C07272=1131.852,246.302,-68.893,-178.601,9.852,149.573
C07273=1131.856,246.053,-68.866,-178.602,9.850,149.573
C07274=1131.860,245.805,-68.838,-178.604,9.848,149.573
C07275=1131.865,245.556,-68.810,-178.605,9.846,149.572
C07276=1131.870,245.308,-68.783,-178.606,9.844,149.572
C07277=1131.874,245.060,-68.754,-178.607,9.842,149.572
C07278=1131.878,244.811,-68.727,-178.609,9.840,149.572
C07279=1131.882,244.563,-68.699,-178.610,9.837,149.572
C07280=1131.887,244.314,-68.672,-178.612,9.835,149.572
C07281=1131.891,244.066,-68.644,-178.613,9.834,149.572
C07282=1131.895,243.818,-68.616,-178.615,9.831,149.572
C07283=1131.900,243.569,-68.589,-178.617,9.829,149.571
C07284=1131.904,243.321,-68.561,-178.618,9.827,149.571
C07285=1131.909,243.072,-68.533,-178.620,9.825,149.571
C07286=1131.913,242.824,-68.506,-178.622,9.822,149.571
C07287=1131.918,242.575,-68.479,-178.623,9.820,149.571
C07288=1131.921,242.327,-68.450,-178.625,9.819,149.571
C07289=1131.926,242.078,-68.423,-178.627,9.816,149.571
C07290=1131.930,241.830,-68.396,-178.629,9.814,149.571
C07291=1131.934,241.581,-68.368,-178.631,9.812,149.571
C07292=1131.939,241.333,-68.340,-178.633,9.809,149.571
C07293=1131.943,241.085,-68.313,-178.635,9.807,149.571
C07294=1131.947,240.836,-68.285,-178.638,9.804,149.571
C07295=1131.952,240.588,-68.258,-178.639,9.802,149.571
C07296=1131.956,240.374,-68.234,-178.641,9.801,149.571
C07297=1131.959,240.159,-68.210,-178.643,9.799,149.571
C07298=1131.964,239.946,-68.186,-178.645,9.796,149.571
C07299=1131.967,239.732,-68.163,-178.647,9.794,149.571
C07300=1131.970,239.517,-68.140,-178.649,9.792,149.571
C07301=1131.974,239.303,-68.116,-178.651,9.790,149.571
C07302=1131.978,239.090,-68.093,-178.653,9.788,149.571
C07303=1131.982,238.876,-68.068,-178.656,9.786,149.571
C07304=1131.986,238.626,-68.041,-178.658,9.783,149.571
C07305=1131.991,238.378,-68.014,-178.661,9.781,149.571
C07306=1131.995,238.130,-67.986,-178.663,9.779,149.572
C07307=1132.000,237.881,-67.959,-178.665,9.775,149.572
C07308=1132.003,237.633,-67.932,-178.668,9.773,149.572
C07309=1132.008,237.385,-67.904,-178.671,9.771,149.572
C07310=1132.012,237.136,-67.877,-178.674,9.768,149.572
C07311=1132.017,236.888,-67.850,-178.677,9.765,149.572
C07312=1132.022,236.639,-67.823,-178.679,9.763,149.572
C07313=1132.025,236.391,-67.795,-178.681,9.760,149.572
C07314=1132.030,236.142,-67.768,-178.684,9.757,149.572
C07315=1132.035,235.894,-67.741,-178.687,9.755,149.572
C07316=1132.039,235.645,-67.714,-178.690,9.752,149.572
C07317=1132.043,235.397,-67.686,-178.693,9.749,149.573
C07318=1132.047,235.148,-67.659,-178.696,9.746,149.573
C07319=1132.052,234.900,-67.632,-178.700,9.743,149.573
C07320=1132.056,234.651,-67.605,-178.703,9.740,149.573
C07321=1132.061,234.403,-67.578,-178.706,9.737,149.573
C07322=1132.065,234.154,-67.551,-178.709,9.735,149.573
C07323=1132.069,233.906,-67.524,-178.713,9.732,149.574
C07324=1132.074,233.657,-67.497,-178.715,9.729,149.574
C07325=1132.078,233.409,-67.470,-178.719,9.725,149.574
C07326=1132.083,233.161,-67.442,-178.722,9.722,149.574
C07327=1132.087,232.912,-67.415,-178.726,9.719,149.574
C07328=1132.091,232.664,-67.389,-178.729,9.717,149.574
C07329=1132.095,232.415,-67.361,-178.733,9.713,149.574
C07330=1132.100,232.166,-67.334,-178.735,9.710,149.575
C07331=1132.104,231.918,-67.308,-178.739,9.707,149.575
C07332=1132.108,231.670,-67.281,-178.743,9.704,149.575
C07333=1132.113,231.421,-67.254,-178.747,9.700,149.575
C07334=1132.118,231.172,-67.227,-178.750,9.697,149.575
C07335=1132.122,230.924,-67.201,-178.753,9.694,149.575
C07336=1132.127,230.675,-67.174,-178.757,9.691,149.576
C07337=1132.131,230.427,-67.147,-178.761,9.687,149.576
C07338=1132.135,230.179,-67.120,-178.765,9.683,149.576
C07339=1132.139,229.929,-67.093,-178.769,9.680,149.576
C07340=1132.143,229.681,-67.066,-178.773,9.676,149.576
C07341=1132.148,229.432,-67.040,-178.777,9.673,149.577
C07342=1132.153,229.184,-67.013,-178.781,9.669,149.577
C07343=1132.157,228.935,-66.987,-178.784,9.665,149.577
C07344=1132.161,228.687,-66.959,-178.788,9.662,149.577
C07345=1132.166,228.438,-66.934,-178.792,9.659,149.577
C07346=1132.170,228.190,-66.907,-178.796,9.655,149.577
C07347=1132.174,227.941,-66.880,-178.799,9.652,149.578
C07348=1132.179,227.692,-66.854,-178.803,9.648,149.578
C07349=1132.184,227.444,-66.827,-178.806,9.644,149.578
C07350=1132.188,227.196,-66.800,-178.810,9.641,149.578
C07351=1132.193,226.947,-66.774,-178.813,9.637,149.578
C07352=1132.197,226.733,-66.751,-178.816,9.634,149.578
C07353=1132.200,226.519,-66.728,-178.820,9.631,149.578
C07354=1132.204,226.305,-66.705,-178.822,9.628,149.578
C07355=1132.207,226.090,-66.683,-178.825,9.625,149.578
C07356=1132.211,225.877,-66.661,-178.828,9.622,149.578
C07357=1132.215,225.662,-66.637,-178.831,9.619,149.578
C07358=1132.219,225.448,-66.615,-178.833,9.616,149.578
C07359=1132.222,225.234,-66.592,-178.836,9.614,149.578
C07360=1132.227,224.985,-66.565,-178.840,9.610,149.578
C07361=1132.231,224.736,-66.539,-178.843,9.606,149.579
C07362=1132.236,224.487,-66.513,-178.846,9.603,149.578
C07363=1132.241,224.240,-66.487,-178.849,9.600,149.579
C07364=1132.245,223.991,-66.461,-178.852,9.596,149.579
C07365=1132.250,223.742,-66.434,-178.855,9.593,149.579
C07366=1132.254,223.494,-66.408,-178.858,9.590,149.579
C07367=1132.258,223.245,-66.382,-178.861,9.586,149.578
C07368=1132.263,222.996,-66.356,-178.864,9.583,149.579
C07369=1132.267,222.747,-66.330,-178.867,9.579,149.579
C07370=1132.271,222.499,-66.303,-178.870,9.576,149.578
C07371=1132.277,222.251,-66.277,-178.873,9.572,149.578
C07372=1132.281,222.002,-66.252,-178.875,9.569,149.578
C07373=1132.285,221.754,-66.225,-178.878,9.566,149.578
C07374=1132.290,221.505,-66.199,-178.881,9.563,149.578
C07375=1132.294,221.256,-66.173,-178.884,9.560,149.578
C07376=1132.298,221.007,-66.147,-178.887,9.556,149.578
C07377=1132.303,220.760,-66.121,-178.889,9.553,149.578
C07378=1132.308,220.511,-66.095,-178.892,9.550,149.578
C07379=1132.312,220.262,-66.069,-178.894,9.547,149.578
C07380=1132.316,220.013,-66.043,-178.897,9.544,149.578
C07381=1132.320,219.765,-66.017,-178.899,9.541,149.578
C07382=1132.325,219.517,-65.992,-178.902,9.538,149.578
C07383=1132.330,219.268,-65.965,-178.904,9.534,149.578
C07384=1132.334,219.019,-65.939,-178.906,9.531,149.578
C07385=1132.338,218.770,-65.914,-178.909,9.528,149.578
C07386=1132.342,218.521,-65.888,-178.911,9.525,149.577
C07387=1132.347,218.273,-65.863,-178.913,9.523,149.577
C07388=1132.351,218.025,-65.836,-178.915,9.519,149.577
C07389=1132.356,217.776,-65.810,-178.918,9.516,149.577
C07390=1132.360,217.527,-65.784,-178.920,9.513,149.577
C07391=1132.365,217.279,-65.759,-178.922,9.511,149.577
C07392=1132.369,217.030,-65.733,-178.924,9.507,149.577
C07393=1132.374,216.781,-65.707,-178.926,9.505,149.577
C07394=1132.378,216.532,-65.681,-178.928,9.501,149.576
C07395=1132.383,216.284,-65.656,-178.930,9.499,149.576
C07396=1132.387,216.036,-65.630,-178.933,9.496,149.576
C07397=1132.391,215.787,-65.604,-178.934,9.493,149.576
C07398=1132.395,215.538,-65.579,-178.937,9.490,149.576
C07399=1132.401,215.289,-65.553,-178.938,9.487,149.576
C07400=1132.405,215.041,-65.527,-178.940,9.485,149.576
C07401=1132.409,214.792,-65.501,-178.942,9.482,149.575
C07402=1132.414,214.544,-65.476,-178.944,9.479,149.575
C07403=1132.418,214.295,-65.450,-178.946,9.477,149.575
C07404=1132.423,214.046,-65.424,-178.948,9.474,149.575
C07405=1132.427,213.797,-65.399,-178.949,9.472,149.575
C07406=1132.432,213.549,-65.373,-178.952,9.468,149.575
C07407=1132.436,213.300,-65.348,-178.953,9.466,149.575
C07408=1132.440,213.087,-65.326,-178.954,9.464,149.574
C07409=1132.443,212.872,-65.304,-178.955,9.462,149.574
C07410=1132.448,212.657,-65.281,-178.957,9.460,149.574
C07411=1132.451,212.443,-65.260,-178.958,9.458,149.574
C07412=1132.456,212.229,-65.238,-178.959,9.456,149.574
C07413=1132.459,212.014,-65.216,-178.960,9.453,149.574
C07414=1132.463,211.800,-65.194,-178.962,9.452,149.574
C07415=1132.467,211.586,-65.172,-178.963,9.449,149.574
C07416=1132.471,211.337,-65.146,-178.965,9.447,149.573
C07417=1132.476,211.088,-65.120,-178.967,9.444,149.573
C07418=1132.481,210.840,-65.095,-178.969,9.442,149.573
C07419=1132.485,210.591,-65.070,-178.970,9.439,149.573
C07420=1132.489,210.343,-65.045,-178.972,9.437,149.573
C07421=1132.493,210.094,-65.019,-178.974,9.435,149.573
C07422=1132.498,209.845,-64.994,-178.976,9.432,149.573
C07423=1132.502,209.597,-64.968,-178.978,9.430,149.573
C07424=1132.507,209.348,-64.943,-178.980,9.427,149.573
C07425=1132.511,209.099,-64.917,-178.982,9.425,149.573
C07426=1132.516,208.851,-64.892,-178.984,9.422,149.573
C07427=1132.521,208.601,-64.867,-178.987,9.419,149.573
C07428=1132.525,208.353,-64.842,-178.988,9.417,149.573
C07429=1132.530,208.104,-64.816,-178.991,9.415,149.573
C07430=1132.534,207.856,-64.790,-178.993,9.412,149.573
C07431=1132.539,207.607,-64.766,-178.995,9.410,149.573
C07432=1132.542,207.358,-64.740,-178.998,9.407,149.573
C07433=1132.547,207.110,-64.715,-179.001,9.404,149.573
C07434=1132.552,206.861,-64.690,-179.003,9.402,149.573
C07435=1132.557,206.613,-64.665,-179.006,9.399,149.573
C07436=1132.561,206.363,-64.640,-179.008,9.396,149.573
C07437=1132.565,206.115,-64.614,-179.011,9.393,149.573
C07438=1132.569,205.867,-64.589,-179.014,9.390,149.573
C07439=1132.574,205.617,-64.564,-179.016,9.387,149.573
C07440=1132.579,205.369,-64.539,-179.019,9.385,149.573
C07441=1132.583,205.120,-64.514,-179.022,9.382,149.573
C07442=1132.588,204.872,-64.488,-179.025,9.379,149.573
C07443=1132.592,204.623,-64.464,-179.028,9.376,149.573
C07444=1132.597,204.375,-64.438,-179.031,9.373,149.574
C07445=1132.601,204.125,-64.413,-179.034,9.370,149.574
C07446=1132.606,203.877,-64.388,-179.037,9.367,149.574
C07447=1132.610,203.628,-64.363,-179.040,9.364,149.574
C07448=1132.615,203.380,-64.338,-179.043,9.361,149.574
C07449=1132.619,203.130,-64.313,-179.046,9.358,149.574
C07450=1132.624,202.882,-64.288,-179.049,9.354,149.574
C07451=1132.628,202.633,-64.263,-179.052,9.352,149.574
C07452=1132.633,202.384,-64.239,-179.056,9.348,149.574
C07453=1132.637,202.136,-64.213,-179.059,9.345,149.575
C07454=1132.642,201.887,-64.189,-179.063,9.342,149.575
C07455=1132.646,201.638,-64.164,-179.066,9.339,149.575
C07456=1132.650,201.390,-64.139,-179.069,9.336,149.575
C07457=1132.655,201.141,-64.114,-179.073,9.333,149.575
C07458=1132.660,200.892,-64.089,-179.077,9.329,149.576
C07459=1132.664,200.644,-64.064,-179.080,9.326,149.576
C07460=1132.669,200.395,-64.039,-179.084,9.322,149.576
C07461=1132.673,200.146,-64.015,-179.087,9.319,149.576
C07462=1132.678,199.897,-63.990,-179.091,9.315,149.576
C07463=1132.683,199.648,-63.966,-179.095,9.312,149.576
C07464=1132.686,199.434,-63.944,-179.099,9.308,149.577
C07465=1132.690,199.220,-63.923,-179.101,9.306,149.577
C07466=1132.694,199.006,-63.902,-179.105,9.302,149.577
C07467=1132.698,198.791,-63.881,-179.108,9.299,149.577
C07468=1132.702,198.577,-63.859,-179.112,9.296,149.577
C07469=1132.706,198.362,-63.838,-179.115,9.293,149.577
C07470=1132.710,198.148,-63.817,-179.118,9.290,149.577
C07471=1132.713,197.933,-63.796,-179.122,9.286,149.578
C07472=1132.718,197.684,-63.771,-179.125,9.283,149.578
C07473=1132.722,197.436,-63.747,-179.130,9.278,149.578
C07474=1132.728,197.187,-63.722,-179.134,9.274,149.578
C07475=1132.731,196.938,-63.698,-179.138,9.271,149.578
C07476=1132.736,196.689,-63.674,-179.142,9.267,149.578
C07477=1132.741,196.441,-63.649,-179.146,9.262,149.579
C07478=1132.745,196.192,-63.625,-179.150,9.259,149.579
C07479=1132.750,195.943,-63.600,-179.151,9.256,149.579
C07480=1132.754,195.694,-63.576,-179.153,9.253,149.578
C07481=1132.759,195.446,-63.552,-179.155,9.251,149.578
C07482=1132.763,195.197,-63.527,-179.155,9.249,149.578
C07483=1132.768,194.948,-63.503,-179.157,9.246,149.578
C07484=1132.772,194.699,-63.479,-179.158,9.244,149.578
C07485=1132.777,194.450,-63.454,-179.160,9.241,149.578
C07486=1132.781,194.201,-63.430,-179.162,9.239,149.577
C07487=1132.786,193.953,-63.406,-179.164,9.236,149.577
C07488=1132.791,193.704,-63.381,-179.165,9.234,149.577
C07489=1132.794,193.455,-63.357,-179.167,9.231,149.577
C07490=1132.799,193.207,-63.333,-179.168,9.229,149.577
C07491=1132.804,192.957,-63.309,-179.170,9.226,149.577
C07492=1132.809,192.709,-63.285,-179.172,9.224,149.576
C07493=1132.813,192.461,-63.261,-179.174,9.221,149.576
C07494=1132.818,192.211,-63.236,-179.175,9.219,149.576
C07495=1132.822,191.963,-63.212,-179.177,9.216,149.576
C07496=1132.827,191.714,-63.188,-179.179,9.214,149.576
C07497=1132.831,191.465,-63.164,-179.180,9.211,149.576
C07498=1132.836,191.217,-63.140,-179.183,9.208,149.576
C07499=1132.840,190.967,-63.115,-179.185,9.206,149.576
C07500=1132.845,190.718,-63.092,-179.186,9.203,149.576
C07501=1132.850,190.470,-63.067,-179.188,9.201,149.576
C07502=1132.854,190.221,-63.043,-179.191,9.198,149.575
C07503=1132.859,189.972,-63.020,-179.193,9.195,149.575
C07504=1132.863,189.723,-62.995,-179.195,9.192,149.575
C07505=1132.867,189.475,-62.971,-179.197,9.190,149.575
C07506=1132.873,189.225,-62.947,-179.200,9.187,149.575
C07507=1132.877,188.977,-62.923,-179.201,9.184,149.575
C07508=1132.881,188.729,-62.899,-179.204,9.181,149.575
C07509=1132.886,188.479,-62.876,-179.205,9.179,149.575
C07510=1132.890,188.230,-62.851,-179.208,9.175,149.575
C07511=1132.895,187.982,-62.827,-179.210,9.173,149.575
C07512=1132.900,187.733,-62.803,-179.213,9.170,149.575
C07513=1132.904,187.484,-62.779,-179.215,9.167,149.575
C07514=1132.909,187.235,-62.756,-179.217,9.165,149.575
C07515=1132.913,186.987,-62.732,-179.220,9.162,149.575
C07516=1132.918,186.738,-62.708,-179.222,9.159,149.575
C07517=1132.923,186.489,-62.684,-179.225,9.156,149.575
C07518=1132.927,186.240,-62.659,-179.227,9.153,149.575
C07519=1132.931,185.991,-62.636,-179.230,9.149,149.575
C07520=1132.935,185.776,-62.615,-179.232,9.147,149.575
C07521=1132.939,185.563,-62.595,-179.234,9.145,149.575
C07522=1132.943,185.348,-62.575,-179.237,9.142,149.575
C07523=1132.947,185.133,-62.555,-179.239,9.140,149.575
C07524=1132.951,184.918,-62.534,-179.241,9.137,149.575
C07525=1132.955,184.704,-62.513,-179.243,9.135,149.575
C07526=1132.959,184.489,-62.492,-179.246,9.132,149.575
C07527=1132.962,184.275,-62.472,-179.248,9.129,149.575
C07528=1132.967,184.026,-62.449,-179.250,9.126,149.575
C07529=1132.972,183.776,-62.425,-179.254,9.123,149.575
C07530=1132.977,183.528,-62.401,-179.256,9.119,149.575
C07531=1132.981,183.279,-62.377,-179.259,9.116,149.575
C07532=1132.986,183.031,-62.353,-179.262,9.114,149.575
C07533=1132.991,182.782,-62.330,-179.265,9.110,149.575
C07534=1132.995,182.533,-62.307,-179.268,9.107,149.575
C07535=1132.999,182.284,-62.283,-179.271,9.104,149.575
C07536=1133.004,182.035,-62.260,-179.274,9.100,149.575
C07537=1133.008,181.786,-62.236,-179.276,9.097,149.575
C07538=1133.013,181.537,-62.213,-179.280,9.093,149.575
C07539=1133.017,181.289,-62.189,-179.282,9.090,149.575
C07540=1133.022,181.040,-62.166,-179.286,9.087,149.575
C07541=1133.027,180.791,-62.142,-179.289,9.083,149.575
C07542=1133.032,180.542,-62.119,-179.292,9.080,149.575
C07543=1133.036,180.293,-62.095,-179.295,9.076,149.575
C07544=1133.041,180.044,-62.071,-179.298,9.072,149.575
C07545=1133.045,179.795,-62.048,-179.301,9.070,149.576
C07546=1133.049,179.547,-62.025,-179.305,9.066,149.576
C07547=1133.054,179.298,-62.002,-179.308,9.062,149.576
C07548=1133.059,179.049,-61.979,-179.311,9.059,149.576
C07549=1133.064,178.800,-61.956,-179.313,9.056,149.575
C07550=1133.069,178.551,-61.932,-179.315,9.053,149.575
C07551=1133.073,178.303,-61.908,-179.317,9.050,149.575
C07552=1133.077,178.054,-61.885,-179.319,9.048,149.575
C07553=1133.082,177.805,-61.862,-179.321,9.044,149.575
C07554=1133.086,177.556,-61.839,-179.324,9.041,149.575
C07555=1133.091,177.307,-61.815,-179.325,9.039,149.575
C07556=1133.096,177.058,-61.792,-179.328,9.036,149.575
C07557=1133.100,176.809,-61.769,-179.330,9.032,149.575
C07558=1133.104,176.560,-61.746,-179.332,9.030,149.575
C07559=1133.109,176.311,-61.722,-179.334,9.027,149.574
C07560=1133.114,176.063,-61.700,-179.337,9.024,149.574
C07561=1133.118,175.814,-61.677,-179.338,9.021,149.574
C07562=1133.123,175.565,-61.653,-179.341,9.018,149.574
C07563=1133.128,175.316,-61.630,-179.343,9.015,149.574
C07564=1133.132,175.067,-61.608,-179.345,9.012,149.574
C07565=1133.137,174.818,-61.585,-179.347,9.009,149.574
C07566=1133.142,174.569,-61.561,-179.350,9.006,149.574
C07567=1133.147,174.320,-61.538,-179.351,9.003,149.574
C07568=1133.151,174.072,-61.515,-179.354,9.000,149.574
C07569=1133.155,173.823,-61.492,-179.356,8.997,149.574
C07570=1133.160,173.574,-61.469,-179.359,8.994,149.573
C07571=1133.164,173.325,-61.446,-179.360,8.991,149.573
C07572=1133.169,173.075,-61.423,-179.363,8.988,149.573
C07573=1133.174,172.827,-61.400,-179.365,8.985,149.573
C07574=1133.178,172.578,-61.378,-179.368,8.982,149.573
C07575=1133.183,172.329,-61.354,-179.369,8.979,149.573
C07576=1133.188,172.089,-61.332,-179.372,8.976,149.573
C07577=1133.192,171.850,-61.310,-179.374,8.973,149.573
C07578=1133.196,171.610,-61.288,-179.376,8.970,149.573
C07579=1133.201,171.370,-61.266,-179.378,8.967,149.573
C07580=1133.206,171.132,-61.245,-179.381,8.964,149.573
C07581=1133.210,170.892,-61.223,-179.383,8.961,149.573
C07582=1133.214,170.652,-61.201,-179.385,8.958,149.572
C07583=1133.219,170.413,-61.179,-179.387,8.955,149.572
C07584=1133.241,169.216,-61.071,-178.557,7.312,148.954
C07585=1133.249,168.816,-61.036,-178.561,7.308,148.954
C07586=1133.253,168.568,-61.014,-178.565,7.306,148.955
C07587=1133.257,168.318,-60.992,-178.567,7.304,148.955
C07588=1133.263,168.070,-60.969,-178.570,7.301,148.955
C07589=1133.267,167.821,-60.947,-178.573,7.300,148.956
C07590=1133.271,167.571,-60.924,-178.576,7.297,148.956
C07591=1133.277,167.323,-60.902,-178.578,7.295,148.956
C07592=1133.281,167.073,-60.880,-178.582,7.292,148.957
C07593=1133.286,166.825,-60.858,-178.584,7.291,148.957
C07594=1133.290,166.576,-60.836,-178.587,7.288,148.957
C07595=1133.296,166.327,-60.813,-178.590,7.286,148.957
C07596=1133.300,166.078,-60.791,-178.593,7.283,148.958
C07597=1133.305,165.829,-60.770,-178.596,7.282,148.958
C07598=1133.309,165.580,-60.748,-178.599,7.279,148.958
C07599=1133.314,165.332,-60.725,-178.602,7.277,148.959
C07600=1133.319,165.082,-60.703,-178.604,7.274,148.959
C07601=1133.323,164.833,-60.681,-178.607,7.273,148.959
C07602=1133.328,164.584,-60.659,-178.610,7.270,148.960
C07603=1133.333,164.335,-60.637,-178.613,7.268,148.960
C07604=1133.337,164.086,-60.615,-178.616,7.266,148.960
C07605=1133.342,163.837,-60.593,-178.619,7.264,148.960
C07606=1133.347,163.588,-60.571,-178.621,7.262,148.961
C07607=1133.352,163.339,-60.549,-178.624,7.259,148.961
C07608=1133.356,163.090,-60.527,-178.627,7.258,148.961
C07609=1133.361,162.841,-60.505,-178.630,7.255,148.961
C07610=1133.365,162.592,-60.483,-178.632,7.253,148.962
C07611=1133.370,162.343,-60.462,-178.636,7.251,148.962
C07612=1133.374,162.094,-60.440,-178.638,7.249,148.962
C07613=1133.379,161.845,-60.418,-178.641,7.246,148.963
C07614=1133.384,161.595,-60.395,-178.644,7.244,148.963
C07615=1133.389,161.347,-60.374,-178.647,7.242,148.963
C07616=1133.393,161.097,-60.352,-178.650,7.240,148.964
C07617=1133.398,160.849,-60.330,-178.652,7.238,148.964
C07618=1133.403,160.600,-60.308,-178.656,7.235,148.964
C07619=1133.407,160.351,-60.286,-178.658,7.233,148.964
C07620=1133.412,160.102,-60.264,-178.661,7.231,148.965
C07621=1133.416,159.853,-60.242,-178.664,7.229,148.965
C07622=1133.421,159.604,-60.221,-178.667,7.227,148.966
C07623=1133.426,159.356,-60.199,-178.669,7.225,148.966
C07624=1133.431,159.106,-60.178,-178.672,7.223,148.966
C07625=1133.435,158.857,-60.156,-178.675,7.220,148.966
C07626=1133.440,158.608,-60.134,-178.678,7.218,148.967
C07627=1133.445,158.359,-60.112,-178.681,7.216,148.967
C07628=1133.449,158.110,-60.091,-178.684,7.214,148.967
C07629=1133.454,157.860,-60.069,-178.687,7.212,148.968
C07630=1133.458,157.592,-60.046,-178.690,7.210,148.968
C07631=1133.464,157.323,-60.022,-178.692,7.207,148.968
C07632=1133.469,157.053,-60.000,-178.696,7.205,148.969
C07633=1133.474,156.785,-59.976,-178.698,7.203,148.969
C07634=1133.479,156.536,-59.954,-178.702,7.200,148.969
C07635=1133.484,156.287,-59.933,-178.704,7.199,148.970
C07636=1133.488,156.038,-59.911,-178.707,7.197,148.970
C07637=1133.493,155.789,-59.889,-178.710,7.194,148.970
C07638=1133.498,155.540,-59.869,-178.713,7.192,148.971
C07639=1133.502,155.291,-59.847,-178.716,7.190,148.971
C07640=1133.507,155.042,-59.825,-178.718,7.188,148.971
C07641=1133.512,154.793,-59.804,-178.721,7.186,148.972
C07642=1133.517,154.544,-59.783,-178.724,7.184,148.972
C07643=1133.521,154.294,-59.761,-178.727,7.182,148.972
C07644=1133.526,154.045,-59.740,-178.730,7.179,148.972
C07645=1133.530,153.797,-59.718,-178.733,7.177,148.973
C07646=1133.535,153.547,-59.697,-178.735,7.176,148.973
C07647=1133.540,153.299,-59.675,-178.739,7.173,148.974
C07648=1133.545,153.049,-59.654,-178.741,7.171,148.974
C07649=1133.550,152.801,-59.633,-178.744,7.169,148.974
C07650=1133.554,152.551,-59.612,-178.747,7.167,148.975
C07651=1133.558,152.302,-59.590,-178.750,7.165,148.975
C07652=1133.564,152.053,-59.569,-178.753,7.163,148.975
C07653=1133.569,151.804,-59.548,-178.755,7.160,148.975
C07654=1133.573,151.554,-59.526,-178.758,7.159,148.976
C07655=1133.577,151.306,-59.505,-178.761,7.156,148.976
C07656=1133.582,151.057,-59.484,-178.764,7.155,148.977
C07657=1133.587,150.808,-59.463,-178.767,7.153,148.977
C07658=1133.592,150.559,-59.442,-178.769,7.150,148.977
C07659=1133.596,150.309,-59.421,-178.772,7.148,148.977
C07660=1133.601,150.061,-59.399,-178.775,7.147,148.978
C07661=1133.606,149.811,-59.378,-178.778,7.144,148.978
C07662=1133.610,149.563,-59.357,-178.781,7.142,148.979
C07663=1133.616,149.314,-59.336,-178.784,7.140,148.979
C07664=1133.621,149.065,-59.315,-178.786,7.138,148.979
C07665=1133.624,148.816,-59.294,-178.789,7.136,148.980
C07666=1133.629,148.566,-59.273,-178.792,7.134,148.980
C07667=1133.635,148.317,-59.252,-178.795,7.132,148.980
C07668=1133.639,148.069,-59.231,-178.797,7.130,148.980
C07669=1133.644,147.819,-59.210,-178.801,7.127,148.981
C07670=1133.649,147.570,-59.189,-178.803,7.126,148.981
C07671=1133.653,147.321,-59.167,-178.806,7.124,148.982
C07672=1133.658,147.072,-59.146,-178.809,7.121,148.982
C07673=1133.662,146.823,-59.126,-178.812,7.119,148.982
C07674=1133.667,146.574,-59.105,-178.814,7.118,148.983
C07675=1133.673,146.324,-59.084,-178.817,7.116,148.983
C07676=1133.677,146.076,-59.063,-178.820,7.113,148.983
C07677=1133.682,145.827,-59.042,-178.823,7.112,148.984
C07678=1133.686,145.578,-59.022,-178.826,7.110,148.984
C07679=1133.691,145.328,-59.000,-178.829,7.107,148.984
C07680=1133.695,145.079,-58.980,-178.831,7.106,148.985
C07681=1133.700,144.830,-58.958,-178.834,7.104,148.985
C07682=1133.705,144.581,-58.937,-178.838,7.101,148.985
C07683=1133.710,144.332,-58.917,-178.840,7.100,148.986
C07684=1133.715,144.083,-58.896,-178.843,7.098,148.986
C07685=1133.719,143.834,-58.876,-178.846,7.095,148.986
C07686=1133.725,143.585,-58.855,-178.849,7.093,148.987
C07687=1133.729,143.336,-58.834,-178.851,7.092,148.987
C07688=1133.734,143.087,-58.814,-178.854,7.090,148.987
C07689=1133.739,142.837,-58.793,-178.857,7.087,148.988
C07690=1133.743,142.589,-58.773,-178.860,7.086,148.988
C07691=1133.748,142.339,-58.752,-178.863,7.084,148.989
C07692=1133.753,142.090,-58.731,-178.866,7.081,148.989
C07693=1133.757,141.841,-58.709,-178.868,7.079,148.989
C07694=1133.761,141.592,-58.689,-178.871,7.078,148.990
C07695=1133.767,141.342,-58.669,-178.874,7.076,148.990
C07696=1133.771,141.093,-58.648,-178.877,7.074,148.990
C07697=1133.776,140.844,-58.628,-178.880,7.072,148.991
C07698=1133.781,140.595,-58.607,-178.882,7.070,148.991
C07699=1133.785,140.346,-58.586,-178.885,7.067,148.991
C07700=1133.791,140.097,-58.566,-178.888,7.066,148.992
C07701=1133.795,139.848,-58.545,-178.891,7.064,148.992
C07702=1133.799,139.599,-58.525,-178.893,7.062,148.992
C07703=1133.805,139.350,-58.504,-178.897,7.060,148.993
C07704=1133.809,139.101,-58.483,-178.899,7.058,148.993
C07705=1133.814,138.852,-58.463,-178.902,7.056,148.994
C07706=1133.819,138.603,-58.442,-178.905,7.055,148.994
C07707=1133.824,138.354,-58.423,-178.908,7.052,148.994
C07708=1133.828,138.105,-58.402,-178.910,7.050,148.995
C07709=1133.834,137.855,-58.381,-178.913,7.048,148.995
C07710=1133.838,137.606,-58.361,-178.916,7.047,148.995
C07711=1133.843,137.358,-58.341,-178.919,7.044,148.996
C07712=1133.848,137.108,-58.320,-178.922,7.043,148.996
C07713=1133.852,136.859,-58.300,-178.925,7.041,148.996
C07714=1133.857,136.610,-58.280,-178.927,7.039,148.997
C07715=1133.861,136.361,-58.259,-178.931,7.037,148.997
C07716=1133.867,136.112,-58.238,-178.933,7.035,148.997
C07717=1133.871,135.862,-58.219,-178.936,7.033,148.998
C07718=1133.876,135.613,-58.198,-178.938,7.031,148.998
C07719=1133.880,135.364,-58.178,-178.942,7.029,148.999
C07720=1133.886,135.115,-58.158,-178.944,7.027,148.999
C07721=1133.891,134.866,-58.138,-178.947,7.025,148.999
C07722=1133.895,134.617,-58.117,-178.950,7.024,149.000
C07723=1133.900,134.367,-58.098,-178.953,7.021,149.000
C07724=1133.904,134.118,-58.077,-178.956,7.019,149.001
C07725=1133.909,133.869,-58.056,-178.959,7.018,149.001
C07726=1133.914,133.620,-58.037,-178.961,7.016,149.001
C07727=1133.919,133.371,-58.016,-178.964,7.014,149.002
C07728=1133.924,133.122,-57.997,-178.967,7.012,149.002
C07729=1133.928,132.873,-57.977,-178.970,7.010,149.002
C07730=1133.933,132.624,-57.956,-178.972,7.008,149.003
C07731=1133.938,132.374,-57.936,-178.975,7.006,149.003
C07732=1133.943,132.125,-57.916,-178.978,7.005,149.004
C07733=1133.947,131.876,-57.896,-178.981,7.002,149.004
C07734=1133.952,131.608,-57.874,-178.984,7.001,149.004
C07735=1133.958,131.339,-57.853,-178.987,6.998,149.005
C07736=1133.963,131.071,-57.832,-178.990,6.996,149.005
C07737=1133.969,130.802,-57.809,-178.993,6.995,149.005
C07738=1133.973,130.553,-57.790,-178.996,6.992,149.006
C07739=1133.978,130.304,-57.769,-178.999,6.991,149.006
C07740=1133.983,130.054,-57.750,-179.001,6.989,149.007
C07741=1133.987,129.805,-57.730,-179.004,6.987,149.007
C07742=1133.992,129.556,-57.710,-179.007,6.985,149.007
C07743=1133.997,129.307,-57.690,-179.010,6.983,149.008
C07744=1134.002,129.058,-57.670,-179.013,6.981,149.008
C07745=1134.006,128.808,-57.650,-179.016,6.980,149.009
C07746=1134.012,128.559,-57.631,-179.018,6.978,149.009
C07747=1134.016,128.310,-57.611,-179.021,6.976,149.009
C07748=1134.021,128.061,-57.591,-179.024,6.975,149.010
C07749=1134.025,127.812,-57.571,-179.027,6.972,149.010
C07750=1134.031,127.563,-57.551,-179.030,6.970,149.011
C07751=1134.035,127.314,-57.532,-179.033,6.969,149.011
C07752=1134.040,127.065,-57.511,-179.035,6.967,149.011
C07753=1134.044,126.815,-57.492,-179.038,6.965,149.012
C07754=1134.050,126.566,-57.472,-179.040,6.963,149.012
C07755=1134.055,126.317,-57.453,-179.044,6.961,149.012
C07756=1134.059,126.068,-57.432,-179.046,6.959,149.013
C07757=1134.064,125.819,-57.413,-179.049,6.957,149.013
C07758=1134.069,125.569,-57.393,-179.052,6.956,149.014
C07759=1134.074,125.320,-57.374,-179.055,6.954,149.014
C07760=1134.078,125.072,-57.354,-179.057,6.952,149.014
C07761=1134.083,124.822,-57.335,-179.060,6.951,149.015
C07762=1134.088,124.573,-57.315,-179.063,6.948,149.015
C07763=1134.092,124.323,-57.295,-179.066,6.946,149.016
C07764=1134.097,124.075,-57.275,-179.069,6.945,149.016
C07765=1134.102,123.825,-57.256,-179.072,6.943,149.016
C07766=1134.107,123.576,-57.236,-179.074,6.941,149.017
C07767=1134.112,123.327,-57.217,-179.077,6.940,149.017
C07768=1134.116,123.077,-57.198,-179.080,6.938,149.018
C07769=1134.122,122.829,-57.178,-179.083,6.936,149.018
C07770=1134.126,122.579,-57.159,-179.086,6.934,149.018
C07771=1134.131,122.329,-57.139,-179.088,6.932,149.019
C07772=1134.136,122.081,-57.119,-179.091,6.930,149.019
C07773=1134.141,121.832,-57.099,-179.094,6.929,149.020
C07774=1134.145,121.582,-57.080,-179.097,6.927,149.020
C07775=1134.150,121.334,-57.061,-179.099,6.925,149.020
C07776=1134.155,121.084,-57.041,-179.102,6.924,149.021
C07777=1134.160,120.835,-57.022,-179.105,6.921,149.021
C07778=1134.164,120.586,-57.003,-179.108,6.920,149.022
C07779=1134.169,120.336,-56.983,-179.111,6.918,149.022
C07780=1134.174,120.087,-56.964,-179.114,6.916,149.022
C07781=1134.179,119.838,-56.945,-179.116,6.915,149.023
C07782=1134.184,119.589,-56.926,-179.119,6.913,149.023
C07783=1134.188,119.340,-56.906,-179.122,6.911,149.024
C07784=1134.193,119.090,-56.887,-179.125,6.909,149.024
C07785=1134.199,118.841,-56.867,-179.127,6.908,149.024
C07786=1134.203,118.592,-56.848,-179.131,6.905,149.025
C07787=1134.208,118.343,-56.829,-179.133,6.904,149.025
C07788=1134.213,118.093,-56.810,-179.136,6.902,149.026
C07789=1134.218,117.844,-56.791,-179.139,6.900,149.026
C07790=1134.222,117.595,-56.772,-179.142,6.899,149.026
C07791=1134.228,117.346,-56.752,-179.144,6.897,149.027
C07792=1134.232,117.097,-56.733,-179.147,6.895,149.027
C07793=1134.237,116.848,-56.714,-179.150,6.894,149.028
C07794=1134.242,116.598,-56.694,-179.152,6.892,149.028
C07795=1134.247,116.349,-56.676,-179.155,6.890,149.028
C07796=1134.251,116.100,-56.657,-179.158,6.889,149.029
C07797=1134.257,115.851,-56.637,-179.161,6.887,149.029
C07798=1134.261,115.601,-56.618,-179.164,6.884,149.030
C07799=1134.266,115.353,-56.599,-179.167,6.883,149.030
C07800=1134.271,115.102,-56.580,-179.169,6.881,149.030
C07801=1134.276,114.854,-56.561,-179.172,6.879,149.031
C07802=1134.280,114.604,-56.542,-179.175,6.878,149.031
C07803=1134.285,114.356,-56.523,-179.178,6.876,149.032
C07804=1134.290,114.105,-56.504,-179.180,6.874,149.032
C07805=1134.295,113.857,-56.485,-179.183,6.873,149.032
C07806=1134.299,113.607,-56.466,-179.186,6.871,149.033
C07807=1134.305,113.358,-56.446,-179.189,6.870,149.034
C07808=1134.309,113.109,-56.428,-179.192,6.868,149.034
C07809=1134.314,112.860,-56.409,-179.194,6.866,149.034
C07810=1134.319,112.611,-56.390,-179.197,6.865,149.035
C07811=1134.324,112.361,-56.371,-179.200,6.863,149.035
C07812=1134.329,112.112,-56.352,-179.203,6.861,149.036
C07813=1134.334,111.862,-56.334,-179.205,6.860,149.036
C07814=1134.338,111.614,-56.315,-179.208,6.858,149.036
C07815=1134.344,111.365,-56.296,-179.211,6.856,149.037
C07816=1134.348,111.115,-56.277,-179.214,6.854,149.037
C07817=1134.353,110.866,-56.258,-179.217,6.852,149.038
C07818=1134.358,110.616,-56.240,-179.220,6.850,149.038
C07819=1134.363,110.367,-56.220,-179.222,6.849,149.038
C07820=1134.368,110.119,-56.202,-179.225,6.847,149.039
C07821=1134.373,109.869,-56.183,-179.228,6.845,149.039
C07822=1134.377,109.620,-56.164,-179.231,6.844,149.040
C07823=1134.382,109.370,-56.146,-179.233,6.842,149.040
C07824=1134.387,109.121,-56.126,-179.236,6.840,149.040
C07825=1134.392,108.872,-56.108,-179.239,6.839,149.041
C07826=1134.397,108.623,-56.089,-179.242,6.837,149.042
C07827=1134.402,108.373,-56.071,-179.245,6.836,149.042
C07828=1134.406,108.125,-56.052,-179.247,6.834,149.042
C07829=1134.411,107.875,-56.033,-179.250,6.832,149.043
C07830=1134.416,107.625,-56.015,-179.253,6.831,149.043
C07831=1134.421,107.377,-55.996,-179.256,6.829,149.044
C07832=1134.426,107.127,-55.977,-179.258,6.827,149.044
C07833=1134.430,106.878,-55.959,-179.261,6.826,149.044
C07834=1134.436,106.629,-55.940,-179.264,6.824,149.045
C07835=1134.440,106.379,-55.922,-179.267,6.822,149.045
C07836=1134.445,106.130,-55.903,-179.269,6.821,149.046
C07837=1134.451,105.881,-55.885,-179.272,6.819,149.046
C07838=1134.455,105.612,-55.865,-179.275,6.818,149.047
C07839=1134.460,105.344,-55.845,-179.278,6.816,149.047
C07840=1134.466,105.076,-55.825,-179.281,6.813,149.047
C07841=1134.471,104.807,-55.805,-179.284,6.812,149.048
C07842=1134.476,104.558,-55.787,-179.287,6.810,149.048
C07843=1134.480,104.309,-55.768,-179.290,6.809,149.049
C07844=1134.485,104.059,-55.750,-179.293,6.807,149.049
C07845=1134.490,103.810,-55.732,-179.296,6.805,149.050
C07846=1134.496,103.561,-55.712,-179.298,6.804,149.050
C07847=1134.500,103.311,-55.694,-179.301,6.802,149.051
C07848=1134.505,103.062,-55.676,-179.304,6.800,149.051
C07849=1134.510,102.813,-55.658,-179.307,6.799,149.051
C07850=1134.515,102.564,-55.639,-179.309,6.797,149.052
C07851=1134.519,102.314,-55.620,-179.312,6.795,149.052
C07852=1134.524,102.065,-55.602,-179.314,6.795,149.053
C07853=1134.529,101.816,-55.584,-179.317,6.793,149.053
C07854=1134.534,101.567,-55.566,-179.320,6.792,149.054
C07855=1134.539,101.317,-55.548,-179.323,6.790,149.054
C07856=1134.544,101.067,-55.530,-179.326,6.788,149.055
C07857=1134.549,100.819,-55.511,-179.328,6.787,149.055
C07858=1134.554,100.570,-55.493,-179.331,6.785,149.055
C07859=1134.558,100.321,-55.475,-179.334,6.783,149.056
C07860=1134.563,100.071,-55.457,-179.336,6.782,149.056
C07861=1134.568,99.821,-55.438,-179.339,6.780,149.057
C07862=1134.573,99.572,-55.420,-179.342,6.778,149.057
C07863=1134.578,99.323,-55.402,-179.345,6.777,149.058
C07864=1134.583,99.074,-55.384,-179.348,6.775,149.058
C07865=1134.588,98.825,-55.366,-179.351,6.774,149.059
C07866=1134.592,98.575,-55.348,-179.353,6.772,149.059
C07867=1134.597,98.325,-55.330,-179.356,6.770,149.059
C07868=1134.602,98.076,-55.312,-179.359,6.769,149.060
C07869=1134.607,97.827,-55.294,-179.362,6.767,149.060
C07870=1134.612,97.578,-55.276,-179.364,6.765,149.061
C07871=1134.617,97.329,-55.258,-179.367,6.765,149.061
C07872=1134.623,97.079,-55.239,-179.370,6.763,149.062
C07873=1134.627,96.829,-55.221,-179.372,6.761,149.062
C07874=1134.632,96.580,-55.203,-179.375,6.760,149.063
C07875=1134.637,96.331,-55.185,-179.378,6.758,149.063
C07876=1134.642,96.082,-55.167,-179.381,6.756,149.063
C07877=1134.647,95.833,-55.149,-179.383,6.755,149.064
C07878=1134.651,95.584,-55.131,-179.386,6.753,149.064
C07879=1134.656,95.334,-55.113,-179.389,6.752,149.065
C07880=1134.661,95.085,-55.095,-179.392,6.750,149.065
C07881=1134.666,94.836,-55.077,-179.395,6.748,149.066
C07882=1134.671,94.587,-55.059,-179.398,6.747,149.066
C07883=1134.676,94.336,-55.041,-179.400,6.746,149.067
C07884=1134.681,94.087,-55.023,-179.402,6.744,149.067
C07885=1134.686,93.838,-55.005,-179.405,6.743,149.067
C07886=1134.690,93.589,-54.987,-179.408,6.741,149.068
C07887=1134.695,93.340,-54.970,-179.411,6.740,149.068
C07888=1134.700,93.091,-54.952,-179.414,6.738,149.069
C07889=1134.705,92.841,-54.935,-179.417,6.736,149.069
C07890=1134.710,92.592,-54.917,-179.419,6.735,149.070
C07891=1134.715,92.343,-54.899,-179.422,6.733,149.070
C07892=1134.720,92.093,-54.881,-179.425,6.731,149.071
C07893=1134.725,91.844,-54.864,-179.428,6.731,149.071
C07894=1134.730,91.594,-54.846,-179.430,6.729,149.072
C07895=1134.735,91.345,-54.828,-179.433,6.728,149.072
C07896=1134.739,91.096,-54.810,-179.436,6.726,149.072
C07897=1134.745,90.846,-54.792,-179.438,6.724,149.073
C07898=1134.749,90.597,-54.775,-179.441,6.723,149.073
C07899=1134.754,90.348,-54.757,-179.444,6.721,149.074
C07900=1134.759,90.098,-54.740,-179.447,6.720,149.074
C07901=1134.764,89.849,-54.722,-179.449,6.719,149.075
C07902=1134.769,89.600,-54.704,-179.452,6.717,149.075
C07903=1134.774,89.350,-54.687,-179.455,6.715,149.076
C07904=1134.778,89.101,-54.669,-179.458,6.714,149.076
C07905=1134.783,88.852,-54.651,-179.460,6.712,149.076
C07906=1134.788,88.603,-54.634,-179.464,6.711,149.077
C07907=1134.793,88.353,-54.616,-179.466,6.709,149.078
C07908=1134.798,88.104,-54.599,-179.469,6.707,149.078
C07909=1134.803,87.855,-54.581,-179.471,6.707,149.078
C07910=1134.808,87.605,-54.564,-179.474,6.705,149.079
C07911=1134.813,87.356,-54.546,-179.477,6.703,149.079
C07912=1134.818,87.107,-54.528,-179.480,6.702,149.080
C07913=1134.822,86.857,-54.511,-179.483,6.700,149.080
C07914=1134.827,86.608,-54.493,-179.485,6.699,149.081
C07915=1134.833,86.359,-54.477,-179.488,6.698,149.081
C07916=1134.838,86.110,-54.459,-179.490,6.696,149.082
C07917=1134.842,85.860,-54.442,-179.493,6.695,149.082
C07918=1134.847,85.611,-54.424,-179.496,6.693,149.083
C07919=1134.852,85.361,-54.407,-179.499,6.692,149.083
C07920=1134.857,85.112,-54.389,-179.502,6.690,149.083
C07921=1134.862,84.862,-54.372,-179.504,6.688,149.084
C07922=1134.867,84.613,-54.355,-179.507,6.687,149.084
C07923=1134.872,84.364,-54.337,-179.510,6.686,149.085
C07924=1134.876,84.114,-54.320,-179.513,6.684,149.085
C07925=1134.882,83.866,-54.302,-179.515,6.683,149.086
C07926=1134.887,83.616,-54.285,-179.518,6.681,149.086
C07927=1134.892,83.366,-54.269,-179.520,6.680,149.087
C07928=1134.897,83.117,-54.251,-179.523,6.679,149.087
C07929=1134.902,82.867,-54.233,-179.526,6.677,149.088
C07930=1134.906,82.618,-54.216,-179.529,6.676,149.088
C07931=1134.911,82.369,-54.199,-179.532,6.674,149.089
C07932=1134.916,82.120,-54.182,-179.534,6.672,149.089
C07933=1134.921,81.871,-54.164,-179.537,6.672,149.090
C07934=1134.926,81.621,-54.147,-179.540,6.670,149.090
C07935=1134.931,81.371,-54.130,-179.543,6.669,149.091
C07936=1134.936,81.122,-54.113,-179.545,6.667,149.091
C07937=1134.940,80.873,-54.096,-179.548,6.665,149.091
C07938=1134.946,80.624,-54.079,-179.551,6.665,149.092
C07939=1134.951,80.374,-54.062,-179.553,6.663,149.093
C07940=1134.955,80.125,-54.044,-179.556,6.661,149.093
C07941=1134.961,79.875,-54.027,-179.559,6.660,149.093
C07942=1134.966,79.607,-54.009,-179.562,6.658,149.094
C07943=1134.971,79.338,-53.991,-179.565,6.657,149.094
C07944=1134.976,79.070,-53.972,-179.568,6.655,149.095
C07945=1134.982,78.802,-53.954,-179.571,6.654,149.096
C07946=1134.987,78.552,-53.937,-179.574,6.652,149.096
C07947=1134.992,78.302,-53.920,-179.576,6.651,149.096
C07948=1134.997,78.054,-53.903,-179.578,6.650,149.097
C07949=1135.002,77.804,-53.886,-179.581,6.648,149.097
C07950=1135.007,77.555,-53.869,-179.584,6.647,149.098
C07951=1135.011,77.305,-53.852,-179.587,6.646,149.098
C07952=1135.017,77.056,-53.835,-179.589,6.644,149.099
C07953=1135.022,76.807,-53.818,-179.592,6.643,149.099
C07954=1135.026,76.557,-53.802,-179.595,6.641,149.100
C07955=1135.031,76.307,-53.784,-179.598,6.640,149.100
C07956=1135.036,76.059,-53.767,-179.600,6.639,149.101
C07957=1135.041,75.809,-53.750,-179.603,6.637,149.101
C07958=1135.046,75.560,-53.734,-179.606,6.636,149.102
C07959=1135.051,75.310,-53.716,-179.609,6.634,149.102
C07960=1135.056,75.061,-53.700,-179.611,6.633,149.103
C07961=1135.061,74.812,-53.683,-179.614,6.632,149.103
C07962=1135.066,74.562,-53.666,-179.617,6.630,149.104
C07963=1135.071,74.313,-53.650,-179.619,6.629,149.104
C07964=1135.076,74.063,-53.632,-179.622,6.628,149.105
C07965=1135.081,73.814,-53.616,-179.625,6.626,149.105
C07966=1135.086,73.565,-53.599,-179.627,6.625,149.105
C07967=1135.091,73.315,-53.582,-179.630,6.623,149.106
C07968=1135.095,73.066,-53.566,-179.633,6.623,149.107
C07969=1135.100,72.817,-53.549,-179.636,6.621,149.107
C07970=1135.106,72.567,-53.532,-179.638,6.619,149.107
C07971=1135.110,72.318,-53.515,-179.641,6.618,149.108
C07972=1135.116,72.068,-53.500,-179.644,6.617,149.109
C07973=1135.121,71.819,-53.482,-179.646,6.616,149.109
C07974=1135.125,71.569,-53.466,-179.649,6.614,149.109
C07975=1135.130,71.320,-53.450,-179.652,6.612,149.110
C07976=1135.136,71.071,-53.432,-179.654,6.611,149.110
C07977=1135.140,70.821,-53.416,-179.657,6.610,149.111
C07978=1135.145,70.572,-53.399,-179.660,6.608,149.111
C07979=1135.150,70.323,-53.382,-179.662,6.608,149.112
C07980=1135.156,70.073,-53.366,-179.665,6.606,149.112
C07981=1135.160,69.824,-53.350,-179.668,6.605,149.113
C07982=1135.165,69.574,-53.333,-179.671,6.603,149.113
C07983=1135.170,69.325,-53.316,-179.673,6.602,149.114
C07984=1135.175,69.076,-53.300,-179.676,6.601,149.114
C07985=1135.180,68.826,-53.284,-179.679,6.599,149.115
C07986=1135.185,68.577,-53.267,-179.681,6.598,149.115
C07987=1135.190,68.327,-53.250,-179.684,6.597,149.116
C07988=1135.195,68.078,-53.234,-179.687,6.595,149.116
C07989=1135.200,67.828,-53.218,-179.690,6.594,149.117
C07990=1135.205,67.579,-53.201,-179.692,6.593,149.117
C07991=1135.209,67.330,-53.185,-179.695,6.591,149.118
C07992=1135.215,67.081,-53.168,-179.698,6.590,149.118
C07993=1135.220,66.831,-53.152,-179.700,6.589,149.119
C07994=1135.225,66.581,-53.135,-179.703,6.588,149.119
C07995=1135.230,66.332,-53.119,-179.706,6.586,149.120
C07996=1135.234,66.082,-53.103,-179.708,6.585,149.120
C07997=1135.239,65.833,-53.087,-179.711,6.584,149.121
C07998=1135.244,65.584,-53.070,-179.714,6.582,149.121
C07999=1135.250,65.334,-53.054,-179.716,6.581,149.122
C08000=1135.255,65.085,-53.037,-179.719,6.580,149.122
C08001=1135.260,64.836,-53.021,-179.722,6.578,149.123
C08002=1135.264,64.586,-53.005,-179.725,6.577,149.123
C08003=1135.270,64.337,-52.989,-179.727,6.576,149.124
C08004=1135.274,64.087,-52.973,-179.730,6.574,149.124
C08005=1135.279,63.838,-52.956,-179.733,6.573,149.125
C08006=1135.284,63.589,-52.940,-179.735,6.572,149.125
C08007=1135.289,63.339,-52.924,-179.738,6.571,149.126
C08008=1135.294,63.090,-52.907,-179.741,6.569,149.126
C08009=1135.299,62.840,-52.892,-179.743,6.568,149.127
C08010=1135.304,62.591,-52.875,-179.746,6.567,149.127
C08011=1135.310,62.341,-52.859,-179.749,6.565,149.128
C08012=1135.314,62.092,-52.842,-179.751,6.564,149.128
C08013=1135.320,61.842,-52.827,-179.754,6.563,149.129
C08014=1135.324,61.593,-52.810,-179.757,6.561,149.129
C08015=1135.329,61.343,-52.794,-179.759,6.561,149.129
C08016=1135.334,61.094,-52.778,-179.762,6.559,149.130
C08017=1135.339,60.845,-52.762,-179.765,6.558,149.131
C08018=1135.344,60.596,-52.746,-179.767,6.557,149.131
C08019=1135.349,60.346,-52.730,-179.770,6.555,149.131
C08020=1135.354,60.097,-52.714,-179.773,6.555,149.132
C08021=1135.359,59.847,-52.698,-179.775,6.553,149.133
C08022=1135.364,59.597,-52.682,-179.778,6.551,149.133
C08023=1135.369,59.348,-52.665,-179.780,6.551,149.133
C08024=1135.374,59.098,-52.650,-179.784,6.549,149.134
C08025=1135.379,58.850,-52.634,-179.786,6.548,149.135
C08026=1135.384,58.600,-52.618,-179.788,6.547,149.135
C08027=1135.389,58.351,-52.603,-179.792,6.546,149.136
C08028=1135.393,58.101,-52.586,-179.794,6.544,149.136
C08029=1135.399,57.852,-52.570,-179.797,6.543,149.137
C08030=1135.404,57.602,-52.555,-179.799,6.541,149.137
C08031=1135.409,57.353,-52.538,-179.802,6.541,149.138
C08032=1135.414,57.103,-52.522,-179.805,6.539,149.138
C08033=1135.419,56.853,-52.507,-179.808,6.538,149.139
C08034=1135.424,56.604,-52.491,-179.810,6.537,149.139
C08035=1135.429,56.355,-52.475,-179.813,6.536,149.140
C08036=1135.434,56.105,-52.459,-179.816,6.534,149.140
C08037=1135.439,55.856,-52.443,-179.818,6.533,149.141
C08038=1135.444,55.607,-52.427,-179.821,6.532,149.141
C08039=1135.449,55.357,-52.411,-179.823,6.531,149.142
C08040=1135.454,55.108,-52.396,-179.826,6.529,149.142
C08041=1135.459,54.858,-52.380,-179.829,6.528,149.143
C08042=1135.464,54.608,-52.364,-179.831,6.527,149.143
C08043=1135.469,54.359,-52.348,-179.834,6.526,149.144
C08044=1135.475,54.110,-52.332,-179.836,6.525,149.144
C08045=1135.479,53.860,-52.317,-179.840,6.524,149.145
C08046=1135.484,53.592,-52.300,-179.842,6.522,149.145
C08047=1135.490,53.323,-52.283,-179.845,6.520,149.146
C08048=1135.495,53.055,-52.266,-179.848,6.520,149.146
C08049=1135.501,52.786,-52.250,-179.850,6.518,149.147
C08050=1135.506,52.537,-52.233,-179.854,6.517,149.147
C08051=1135.510,52.287,-52.218,-179.856,6.516,149.148
C08052=1135.516,52.038,-52.202,-179.859,6.514,149.148
C08053=1135.521,51.788,-52.187,-179.862,6.513,149.149
C08054=1135.526,51.538,-52.171,-179.864,6.512,149.149
C08055=1135.530,51.289,-52.156,-179.867,6.511,149.150
C08056=1135.536,51.040,-52.140,-179.869,6.510,149.150
C08057=1135.541,50.790,-52.125,-179.872,6.509,149.151
C08058=1135.546,50.540,-52.109,-179.874,6.508,149.151
C08059=1135.551,50.291,-52.094,-179.877,6.506,149.152
C08060=1135.556,50.042,-52.078,-179.880,6.505,149.152
C08061=1135.561,49.792,-52.063,-179.882,6.504,149.153
C08062=1135.565,49.542,-52.047,-179.885,6.502,149.153
C08063=1135.571,49.293,-52.032,-179.888,6.502,149.154
C08064=1135.576,49.044,-52.016,-179.891,6.500,149.154
C08065=1135.581,48.794,-52.001,-179.893,6.499,149.155
C08066=1135.586,48.544,-51.985,-179.896,6.498,149.155
C08067=1135.591,48.295,-51.970,-179.899,6.497,149.156
C08068=1135.596,48.046,-51.955,-179.901,6.496,149.157
C08069=1135.601,47.796,-51.939,-179.904,6.494,149.157
C08070=1135.607,47.547,-51.923,-179.906,6.494,149.158
C08071=1135.611,47.297,-51.908,-179.909,6.492,149.158
C08072=1135.616,47.048,-51.892,-179.911,6.491,149.159
C08073=1135.621,46.798,-51.877,-179.915,6.490,149.159
C08074=1135.626,46.549,-51.862,-179.917,6.489,149.160
C08075=1135.631,46.300,-51.846,-179.919,6.487,149.160
C08076=1135.635,46.050,-51.831,-179.922,6.487,149.161
C08077=1135.641,45.800,-51.816,-179.925,6.485,149.161
C08078=1135.646,45.551,-51.800,-179.928,6.484,149.162
C08079=1135.651,45.302,-51.785,-179.930,6.483,149.162
C08080=1135.657,45.052,-51.770,-179.933,6.482,149.163
C08081=1135.661,44.803,-51.755,-179.935,6.481,149.163
C08082=1135.667,44.554,-51.739,-179.938,6.479,149.164
C08083=1135.671,44.303,-51.725,-179.941,6.479,149.164
C08084=1135.676,44.054,-51.709,-179.943,6.477,149.165
C08085=1135.682,43.805,-51.693,-179.946,6.476,149.165
C08086=1135.686,43.555,-51.678,-179.949,6.475,149.166
C08087=1135.692,43.306,-51.663,-179.951,6.474,149.166
C08088=1135.697,43.056,-51.649,-179.954,6.473,149.167
C08089=1135.702,42.807,-51.633,-179.956,6.472,149.167
C08090=1135.707,42.558,-51.618,-179.959,6.471,149.168
C08091=1135.712,42.308,-51.602,-179.961,6.470,149.168
C08092=1135.716,42.058,-51.588,-179.964,6.468,149.169
C08093=1135.722,41.809,-51.572,-179.967,6.468,149.169
C08094=1135.726,41.560,-51.557,-179.969,6.466,149.170
C08095=1135.732,41.310,-51.542,-179.972,6.465,149.170
C08096=1135.737,41.060,-51.527,-179.975,6.464,149.171
C08097=1135.742,40.811,-51.512,-179.977,6.463,149.171
C08098=1135.747,40.561,-51.497,-179.980,6.461,149.172
C08099=1135.753,40.312,-51.482,-179.982,6.461,149.173
C08100=1135.757,40.063,-51.467,-179.985,6.459,149.173
C08101=1135.762,39.813,-51.453,-179.987,6.459,149.174
C08102=1135.768,39.564,-51.437,-179.991,6.457,149.174
C08103=1135.772,39.314,-51.422,-179.993,6.456,149.175
C08104=1135.777,39.064,-51.407,-179.995,6.455,149.175
C08105=1135.782,38.815,-51.392,-179.998,6.454,149.176
C08106=1135.788,38.565,-51.377,179.999,6.453,149.176
C08107=1135.792,38.316,-51.362,179.997,6.452,149.177
C08108=1135.797,38.066,-51.348,179.994,6.451,149.177
C08109=1135.803,37.817,-51.332,179.992,6.450,149.178
C08110=1135.807,37.567,-51.317,179.989,6.448,149.178
C08111=1135.812,37.318,-51.303,179.986,6.448,149.179
C08112=1135.818,37.068,-51.287,179.983,6.446,149.179
C08113=1135.823,36.819,-51.273,179.981,6.445,149.180
C08114=1135.828,36.569,-51.257,179.978,6.444,149.180
C08115=1135.833,36.320,-51.243,179.976,6.443,149.181
C08116=1135.838,36.070,-51.228,179.973,6.442,149.181
C08117=1135.843,35.820,-51.213,179.970,6.441,149.182
C08118=1135.848,35.571,-51.198,179.968,6.440,149.183
C08119=1135.853,35.322,-51.184,179.965,6.439,149.183
C08120=1135.859,35.072,-51.169,179.963,6.437,149.183
C08121=1135.863,34.823,-51.154,179.960,6.437,149.184
C08122=1135.868,34.573,-51.140,179.958,6.436,149.185
C08123=1135.873,34.324,-51.125,179.955,6.434,149.185
C08124=1135.879,34.074,-51.110,179.952,6.434,149.186
C08125=1135.884,33.825,-51.095,179.950,6.432,149.186
C08126=1135.889,33.576,-51.081,179.948,6.431,149.187
C08127=1135.894,33.326,-51.066,179.944,6.430,149.187
C08128=1135.899,33.076,-51.051,179.942,6.429,149.188
C08129=1135.904,32.827,-51.037,179.939,6.428,149.188
C08130=1135.909,32.578,-51.022,179.937,6.427,149.189
C08131=1135.914,32.328,-51.007,179.934,6.426,149.189
C08132=1135.919,32.078,-50.993,179.932,6.425,149.190
C08133=1135.924,31.829,-50.978,179.929,6.424,149.190
C08134=1135.929,31.579,-50.963,179.926,6.423,149.191
C08135=1135.934,31.329,-50.949,179.924,6.422,149.191
C08136=1135.940,31.079,-50.934,179.921,6.421,149.192
C08137=1135.944,30.830,-50.919,179.919,6.420,149.192
C08138=1135.949,30.581,-50.905,179.916,6.418,149.193
C08139=1135.955,30.332,-50.891,179.913,6.418,149.194
C08140=1135.959,30.083,-50.876,179.911,6.417,149.194
C08141=1135.965,29.833,-50.861,179.908,6.415,149.194
C08142=1135.970,29.583,-50.847,179.906,6.415,149.195
C08143=1135.975,29.333,-50.833,179.903,6.413,149.196
C08144=1135.980,29.084,-50.818,179.901,6.412,149.196
C08145=1135.985,28.834,-50.803,179.898,6.411,149.197
C08146=1135.990,28.585,-50.789,179.895,6.410,149.197
C08147=1135.996,28.335,-50.775,179.893,6.410,149.198
C08148=1136.001,28.086,-50.760,179.890,6.408,149.198
C08149=1136.005,27.836,-50.745,179.888,6.407,149.199
C08150=1136.011,27.567,-50.730,179.885,6.406,149.199
C08151=1136.016,27.298,-50.715,179.882,6.405,149.200
C08152=1136.021,27.029,-50.700,179.879,6.404,149.201
C08153=1136.027,26.760,-50.683,179.876,6.403,149.201
C08154=1136.033,26.511,-50.670,179.874,6.402,149.202
C08155=1136.038,26.261,-50.655,179.872,6.401,149.202
C08156=1136.043,26.011,-50.641,179.869,6.400,149.203
C08157=1136.047,25.762,-50.626,179.866,6.399,149.203
C08158=1136.052,25.512,-50.612,179.863,6.398,149.204
C08159=1136.057,25.263,-50.597,179.861,6.397,149.204
C08160=1136.063,25.014,-50.584,179.859,6.396,149.205
C08161=1136.068,24.764,-50.569,179.856,6.395,149.205
C08162=1136.073,24.514,-50.555,179.854,6.394,149.206
C08163=1136.078,24.265,-50.541,179.850,6.393,149.207
C08164=1136.083,24.016,-50.527,179.848,6.392,149.207
C08165=1136.088,23.766,-50.512,179.846,6.391,149.207
C08166=1136.093,23.516,-50.498,179.843,6.390,149.208
C08167=1136.098,23.266,-50.484,179.841,6.389,149.209
C08168=1136.103,23.017,-50.470,179.838,6.388,149.209
C08169=1136.109,22.768,-50.456,179.835,6.387,149.210
C08170=1136.114,22.518,-50.441,179.833,6.386,149.210
C08171=1136.119,22.268,-50.427,179.830,6.384,149.211
C08172=1136.124,22.019,-50.413,179.828,6.384,149.211
C08173=1136.129,21.770,-50.399,179.825,6.383,149.212
C08174=1136.134,21.520,-50.385,179.823,6.382,149.212
C08175=1136.139,21.270,-50.370,179.820,6.381,149.213
C08176=1136.144,21.021,-50.356,179.818,6.380,149.213
C08177=1136.149,20.772,-50.342,179.815,6.379,149.214
C08178=1136.154,20.522,-50.328,179.812,6.378,149.214
C08179=1136.159,20.272,-50.314,179.810,6.377,149.215
C08180=1136.165,20.022,-50.301,179.807,6.376,149.216
C08181=1136.170,19.773,-50.286,179.805,6.375,149.216
C08182=1136.175,19.523,-50.272,179.802,6.374,149.217
C08183=1136.179,19.274,-50.258,179.799,6.373,149.217
C08184=1136.185,19.025,-50.244,179.797,6.373,149.218
C08185=1136.190,18.775,-50.230,179.794,6.371,149.218
C08186=1136.195,18.525,-50.216,179.792,6.371,149.219
C08187=1136.201,18.276,-50.203,179.790,6.370,149.219
C08188=1136.206,18.026,-50.188,179.787,6.368,149.220
C08189=1136.211,17.776,-50.174,179.784,6.368,149.220
C08190=1136.216,17.527,-50.160,179.782,6.367,149.221
C08191=1136.220,17.278,-50.146,179.779,6.365,149.221
C08192=1136.226,17.027,-50.133,179.777,6.365,149.222
C08193=1136.231,16.778,-50.119,179.774,6.364,149.222
C08194=1136.236,16.529,-50.105,179.772,6.362,149.223
C08195=1136.241,16.279,-50.090,179.769,6.362,149.224
C08196=1136.247,16.030,-50.077,179.767,6.361,149.224
C08197=1136.251,15.780,-50.064,179.764,6.360,149.225
C08198=1136.256,15.530,-50.049,179.761,6.359,149.225
C08199=1136.262,15.281,-50.035,179.759,6.358,149.226
C08200=1136.267,15.031,-50.022,179.756,6.357,149.226
C08201=1136.272,14.781,-50.008,179.754,6.356,149.227
C08202=1136.277,14.532,-49.994,179.752,6.355,149.227
C08203=1136.282,14.283,-49.980,179.748,6.354,149.228
C08204=1136.288,14.033,-49.967,179.746,6.353,149.228
C08205=1136.293,13.783,-49.952,179.744,6.353,149.229
C08206=1136.297,13.534,-49.939,179.741,6.351,149.230
C08207=1136.303,13.284,-49.926,179.739,6.351,149.230
C08208=1136.308,13.035,-49.911,179.737,6.350,149.231
C08209=1136.313,12.785,-49.898,179.733,6.349,149.231
C08210=1136.318,12.536,-49.884,179.731,6.348,149.232
C08211=1136.323,12.286,-49.870,179.729,6.347,149.232
C08212=1136.328,12.036,-49.857,179.726,6.346,149.233
C08213=1136.333,11.787,-49.843,179.723,6.345,149.233
C08214=1136.338,11.538,-49.829,179.721,6.344,149.234
C08215=1136.343,11.288,-49.816,179.719,6.344,149.234
C08216=1136.349,11.039,-49.802,179.716,6.342,149.235
C08217=1136.354,10.789,-49.789,179.713,6.342,149.236
C08218=1136.359,10.539,-49.775,179.711,6.341,149.236
C08219=1136.364,10.289,-49.761,179.708,6.339,149.236
C08220=1136.369,10.040,-49.748,179.706,6.339,149.237
C08221=1136.374,9.790,-49.735,179.703,6.338,149.238
C08222=1136.379,9.540,-49.720,179.701,6.337,149.238
C08223=1136.385,9.291,-49.708,179.698,6.336,149.239
C08224=1136.389,9.041,-49.693,179.696,6.335,149.239
C08225=1136.395,8.792,-49.680,179.694,6.334,149.240
C08226=1136.400,8.542,-49.667,179.690,6.333,149.240
C08227=1136.405,8.293,-49.653,179.688,6.332,149.241
C08228=1136.410,8.043,-49.639,179.686,6.331,149.241
C08229=1136.416,7.794,-49.626,179.683,6.331,149.242
C08230=1136.420,7.544,-49.612,179.681,6.329,149.242
C08231=1136.426,7.295,-49.600,179.678,6.329,149.243
C08232=1136.431,7.045,-49.585,179.676,6.328,149.244
C08233=1136.436,6.795,-49.572,179.674,6.327,149.244
C08234=1136.441,6.545,-49.559,179.670,6.326,149.245
C08235=1136.446,6.296,-49.545,179.668,6.325,149.245
C08236=1136.451,6.046,-49.532,179.666,6.325,149.246
C08237=1136.457,5.797,-49.518,179.663,6.324,149.246
C08238=1136.461,5.547,-49.505,179.661,6.322,149.247
C08239=1136.467,5.298,-49.492,179.658,6.322,149.247
C08240=1136.471,5.048,-49.479,179.656,6.321,149.248
C08241=1136.477,4.799,-49.465,179.653,6.320,149.248
C08242=1136.482,4.549,-49.452,179.651,6.319,149.249
C08243=1136.487,4.300,-49.438,179.648,6.318,149.250
C08244=1136.492,4.049,-49.425,179.646,6.318,149.250
C08245=1136.497,3.800,-49.412,179.643,6.316,149.251
C08246=1136.503,3.551,-49.398,179.641,6.316,149.251
C08247=1136.508,3.301,-49.385,179.638,6.315,149.252
C08248=1136.513,3.051,-49.372,179.636,6.314,149.252
C08249=1136.518,2.802,-49.359,179.634,6.314,149.253
C08250=1136.523,2.553,-49.346,179.631,6.312,149.253
C08251=1136.528,2.302,-49.332,179.628,6.312,149.254
C08252=1136.533,2.053,-49.320,179.626,6.311,149.254
C08253=1136.539,1.804,-49.306,179.624,6.310,149.255
C08254=1136.544,1.534,-49.292,179.620,6.309,149.256
C08255=1136.549,1.264,-49.278,179.618,6.308,149.256
C08256=1136.555,0.995,-49.263,179.615,6.307,149.257
C08257=1136.561,0.725,-49.249,179.612,6.306,149.257
C08258=1136.566,0.475,-49.236,179.610,6.305,149.258
C08259=1136.571,0.226,-49.223,179.607,6.304,149.258
C08260=1136.576,-0.023,-49.210,179.605,6.303,149.259
C08261=1136.581,-0.273,-49.197,179.603,6.303,149.260
C08262=1136.587,-0.523,-49.183,179.600,6.302,149.260
C08263=1136.591,-0.773,-49.170,179.598,6.301,149.261
C08264=1136.596,-1.022,-49.158,179.595,6.300,149.261
C08265=1136.602,-1.271,-49.145,179.593,6.299,149.262
C08266=1136.607,-1.521,-49.131,179.590,6.299,149.262
C08267=1136.612,-1.771,-49.118,179.588,6.298,149.263
C08268=1136.618,-2.020,-49.105,179.585,6.297,149.263
C08269=1136.622,-2.270,-49.092,179.583,6.296,149.264
C08270=1136.628,-2.519,-49.079,179.580,6.295,149.264
C08271=1136.633,-2.769,-49.066,179.578,6.295,149.265
C08272=1136.638,-3.019,-49.053,179.576,6.294,149.266
C08273=1136.643,-3.268,-49.040,179.573,6.293,149.266
C08274=1136.649,-3.518,-49.028,179.570,6.292,149.267
C08275=1136.653,-3.768,-49.015,179.568,6.291,149.267
C08276=1136.659,-4.017,-49.001,179.566,6.290,149.268
C08277=1136.664,-4.267,-48.989,179.563,6.290,149.268
C08278=1136.669,-4.517,-48.976,179.561,6.289,149.269
C08279=1136.674,-4.766,-48.963,179.558,6.287,149.269
C08280=1136.680,-5.016,-48.950,179.555,6.287,149.270
C08281=1136.685,-5.265,-48.937,179.553,6.286,149.270
C08282=1136.690,-5.515,-48.924,179.551,6.286,149.271
C08283=1136.695,-5.765,-48.911,179.548,6.285,149.272
C08284=1136.700,-6.014,-48.899,179.546,6.283,149.272
C08285=1136.705,-6.264,-48.886,179.543,6.283,149.273
C08286=1136.711,-6.514,-48.873,179.541,6.282,149.273
C08287=1136.716,-6.763,-48.860,179.539,6.281,149.274
C08288=1136.721,-7.012,-48.847,179.536,6.281,149.274
C08289=1136.725,-7.262,-48.834,179.534,6.280,149.275
C08290=1136.731,-7.512,-48.821,179.531,6.278,149.275
C08291=1136.736,-7.761,-48.809,179.528,6.278,149.276
C08292=1136.741,-8.011,-48.796,179.526,6.277,149.276
C08293=1136.746,-8.261,-48.783,179.524,6.276,149.277
C08294=1136.751,-8.510,-48.770,179.521,6.276,149.278
C08295=1136.757,-8.760,-48.757,179.519,6.275,149.278
C08296=1136.762,-9.009,-48.745,179.516,6.274,149.279
C08297=1136.767,-9.259,-48.732,179.514,6.273,149.279
C08298=1136.772,-9.509,-48.720,179.512,6.272,149.280
C08299=1136.777,-9.758,-48.707,179.509,6.272,149.280
C08300=1136.783,-10.008,-48.694,179.507,6.271,149.281
C08301=1136.788,-10.257,-48.681,179.505,6.270,149.281
C08302=1136.793,-10.508,-48.669,179.501,6.269,149.282
C08303=1136.798,-10.757,-48.656,179.499,6.268,149.283
C08304=1136.803,-11.006,-48.644,179.497,6.268,149.283
C08305=1136.808,-11.256,-48.631,179.494,6.267,149.284
C08306=1136.813,-11.506,-48.618,179.492,6.266,149.284
C08307=1136.819,-11.756,-48.606,179.490,6.266,149.285
C08308=1136.824,-12.005,-48.593,179.487,6.265,149.285
C08309=1136.829,-12.255,-48.581,179.484,6.264,149.286
C08310=1136.834,-12.504,-48.568,179.482,6.263,149.286
C08311=1136.840,-12.753,-48.555,179.480,6.262,149.287
C08312=1136.844,-13.004,-48.543,179.477,6.262,149.287
C08313=1136.849,-13.253,-48.531,179.475,6.261,149.288
C08314=1136.855,-13.502,-48.518,179.473,6.260,149.289
C08315=1136.860,-13.752,-48.506,179.470,6.260,149.289
C08316=1136.865,-14.002,-48.494,179.467,6.258,149.290
C08317=1136.871,-14.251,-48.480,179.465,6.258,149.290
C08318=1136.876,-14.501,-48.467,179.463,6.257,149.291
C08319=1136.881,-14.751,-48.455,179.460,6.256,149.291
C08320=1136.886,-15.001,-48.443,179.458,6.256,149.292
C08321=1136.891,-15.250,-48.430,179.456,6.255,149.292
C08322=1136.897,-15.500,-48.418,179.453,6.254,149.293
C08323=1136.902,-15.749,-48.406,179.451,6.254,149.293
C08324=1136.907,-15.999,-48.394,179.448,6.252,149.294
C08325=1136.912,-16.248,-48.381,179.445,6.252,149.295
C08326=1136.917,-16.498,-48.368,179.443,6.251,149.295
C08327=1136.922,-16.748,-48.356,179.441,6.250,149.296
C08328=1136.927,-16.998,-48.344,179.438,6.250,149.296
C08329=1136.933,-17.247,-48.331,179.436,6.249,149.297
C08330=1136.938,-17.497,-48.319,179.434,6.248,149.297
C08331=1136.943,-17.746,-48.307,179.431,6.248,149.298
C08332=1136.949,-17.996,-48.295,179.429,6.247,149.298
C08333=1136.954,-18.246,-48.282,179.426,6.246,149.299
C08334=1136.959,-18.495,-48.270,179.424,6.245,149.300
C08335=1136.964,-18.745,-48.258,179.422,6.244,149.300
C08336=1136.969,-18.995,-48.246,179.419,6.244,149.301
C08337=1136.974,-19.245,-48.233,179.417,6.243,149.301
C08338=1136.979,-19.494,-48.220,179.415,6.242,149.302
C08339=1136.985,-19.744,-48.208,179.412,6.242,149.302
C08340=1136.990,-19.993,-48.196,179.410,6.241,149.303
C08341=1136.995,-20.243,-48.184,179.408,6.240,149.303
C08342=1137.000,-20.493,-48.171,179.405,6.240,149.304
C08343=1137.006,-20.743,-48.159,179.403,6.239,149.304
C08344=1137.010,-20.992,-48.148,179.400,6.237,149.305
C08345=1137.016,-21.241,-48.136,179.397,6.237,149.306
C08346=1137.021,-21.491,-48.124,179.395,6.236,149.306
C08347=1137.026,-21.741,-48.111,179.393,6.235,149.307
C08348=1137.032,-21.991,-48.099,179.390,6.235,149.307
C08349=1137.037,-22.240,-48.087,179.388,6.234,149.308
C08350=1137.042,-22.490,-48.075,179.386,6.233,149.308
C08351=1137.047,-22.739,-48.062,179.383,6.233,149.309
C08352=1137.053,-22.989,-48.050,179.381,6.232,149.309
C08353=1137.057,-23.239,-48.039,179.379,6.231,149.310
C08354=1137.063,-23.488,-48.026,179.376,6.231,149.311
C08355=1137.068,-23.738,-48.014,179.374,6.230,149.311
C08356=1137.073,-23.988,-48.003,179.372,6.229,149.311
C08357=1137.078,-24.237,-47.990,179.369,6.228,149.312
C08358=1137.084,-24.508,-47.977,179.366,6.227,149.313
C08359=1137.090,-24.777,-47.964,179.364,6.227,149.313
C08360=1137.095,-25.048,-47.951,179.362,6.226,149.314
C08361=1137.101,-25.318,-47.938,179.359,6.226,149.315
C08362=1137.105,-25.567,-47.926,179.357,6.225,149.315
C08363=1137.111,-25.817,-47.914,179.353,6.224,149.316
C08364=1137.117,-26.066,-47.902,179.351,6.223,149.316
C08365=1137.122,-26.316,-47.891,179.349,6.222,149.317
C08366=1137.127,-26.566,-47.878,179.346,6.222,149.317
C08367=1137.132,-26.815,-47.867,179.344,6.221,149.318
C08368=1137.138,-27.065,-47.855,179.342,6.220,149.318
C08369=1137.143,-27.315,-47.842,179.339,6.220,149.319
C08370=1137.148,-27.565,-47.830,179.337,6.219,149.319
C08371=1137.153,-27.814,-47.819,179.335,6.218,149.320
C08372=1137.158,-28.064,-47.807,179.332,6.218,149.321
C08373=1137.163,-28.313,-47.795,179.330,6.217,149.321
C08374=1137.169,-28.563,-47.783,179.328,6.216,149.322
C08375=1137.174,-28.813,-47.771,179.325,6.216,149.322
C08376=1137.179,-29.063,-47.759,179.323,6.215,149.323
C08377=1137.184,-29.313,-47.748,179.321,6.214,149.323
C08378=1137.189,-29.562,-47.735,179.318,6.214,149.324
C08379=1137.194,-29.812,-47.724,179.316,6.213,149.324
C08380=1137.200,-30.061,-47.712,179.314,6.212,149.325
C08381=1137.206,-30.311,-47.700,179.311,6.212,149.326
C08382=1137.210,-30.561,-47.689,179.309,6.211,149.326
C08383=1137.215,-30.810,-47.676,179.307,6.210,149.327
C08384=1137.221,-31.060,-47.665,179.304,6.210,149.327
C08385=1137.226,-31.309,-47.653,179.302,6.209,149.328
C08386=1137.231,-31.559,-47.641,179.300,6.208,149.328
C08387=1137.236,-31.809,-47.629,179.297,6.208,149.329
C08388=1137.241,-32.059,-47.618,179.295,6.207,149.329
C08389=1137.247,-32.308,-47.607,179.293,6.206,149.330
C08390=1137.253,-32.558,-47.595,179.290,6.206,149.330
C08391=1137.257,-32.808,-47.583,179.288,6.205,149.331
C08392=1137.262,-33.057,-47.571,179.286,6.204,149.331
C08393=1137.268,-33.307,-47.559,179.283,6.204,149.332
C08394=1137.273,-33.557,-47.548,179.281,6.203,149.333
C08395=1137.278,-33.807,-47.536,179.279,6.202,149.333
C08396=1137.283,-34.056,-47.525,179.276,6.202,149.334
C08397=1137.289,-34.305,-47.513,179.274,6.201,149.334
C08398=1137.294,-34.555,-47.501,179.272,6.200,149.335
C08399=1137.299,-34.805,-47.490,179.269,6.200,149.335
C08400=1137.304,-35.055,-47.478,179.267,6.199,149.336
C08401=1137.309,-35.305,-47.467,179.265,6.199,149.336
C08402=1137.315,-35.554,-47.455,179.262,6.198,149.337
C08403=1137.320,-35.804,-47.443,179.260,6.197,149.338
C08404=1137.325,-36.053,-47.432,179.258,6.197,149.338
C08405=1137.331,-36.303,-47.420,179.255,6.196,149.339
C08406=1137.335,-36.553,-47.409,179.253,6.195,149.339
C08407=1137.341,-36.802,-47.397,179.251,6.195,149.340
C08408=1137.346,-37.052,-47.386,179.248,6.194,149.340
C08409=1137.351,-37.302,-47.374,179.246,6.193,149.341
C08410=1137.357,-37.552,-47.362,179.244,6.193,149.341
C08411=1137.362,-37.801,-47.351,179.241,6.192,149.342
C08412=1137.368,-38.051,-47.339,179.239,6.191,149.343
C08413=1137.373,-38.301,-47.329,179.237,6.191,149.343
C08414=1137.378,-38.551,-47.317,179.234,6.190,149.344
C08415=1137.383,-38.800,-47.306,179.232,6.189,149.344
C08416=1137.389,-39.050,-47.294,179.229,6.189,149.345
C08417=1137.393,-39.299,-47.283,179.227,6.188,149.345
C08418=1137.399,-39.549,-47.271,179.225,6.188,149.346
C08419=1137.403,-39.799,-47.260,179.222,6.187,149.346
C08420=1137.409,-40.048,-47.248,179.220,6.186,149.347
C08421=1137.414,-40.298,-47.238,179.218,6.186,149.347
C08422=1137.420,-40.548,-47.226,179.215,6.185,149.348
C08423=1137.425,-40.797,-47.215,179.213,6.184,149.348
C08424=1137.431,-41.047,-47.203,179.211,6.184,149.349
C08425=1137.435,-41.297,-47.192,179.208,6.183,149.350
C08426=1137.441,-41.547,-47.180,179.206,6.182,149.350
C08427=1137.446,-41.796,-47.170,179.203,6.182,149.351
C08428=1137.451,-42.046,-47.158,179.201,6.181,149.351
C08429=1137.456,-42.296,-47.146,179.199,6.180,149.352
C08430=1137.461,-42.545,-47.135,179.196,6.180,149.352
C08431=1137.467,-42.795,-47.124,179.194,6.179,149.353
C08432=1137.472,-43.045,-47.113,179.192,6.178,149.353
C08433=1137.477,-43.294,-47.102,179.190,6.177,149.354
C08434=1137.483,-43.544,-47.090,179.187,6.177,149.355
C08435=1137.488,-43.793,-47.079,179.186,6.177,149.355
C08436=1137.493,-44.044,-47.068,179.183,6.176,149.356
C08437=1137.499,-44.293,-47.057,179.181,6.176,149.356
C08438=1137.503,-44.542,-47.045,179.179,6.175,149.357
C08439=1137.509,-44.792,-47.034,179.176,6.174,149.357
C08440=1137.514,-45.042,-47.023,179.174,6.174,149.358
C08441=1137.520,-45.292,-47.011,179.172,6.173,149.358
C08442=1137.524,-45.541,-47.000,179.169,6.172,149.359
C08443=1137.530,-45.791,-46.990,179.167,6.172,149.360
C08444=1137.536,-46.041,-46.978,179.164,6.171,149.360
C08445=1137.540,-46.291,-46.967,179.162,6.170,149.361
C08446=1137.546,-46.540,-46.957,179.160,6.170,149.361
C08447=1137.551,-46.790,-46.945,179.157,6.169,149.362
C08448=1137.556,-47.040,-46.933,179.155,6.168,149.362
C08449=1137.562,-47.289,-46.923,179.153,6.168,149.363
C08450=1137.567,-47.539,-46.911,179.151,6.168,149.363
C08451=1137.572,-47.789,-46.901,179.149,6.167,149.364
C08452=1137.577,-48.038,-46.890,179.147,6.167,149.364
C08453=1137.583,-48.288,-46.878,179.144,6.166,149.365
C08454=1137.588,-48.538,-46.867,179.142,6.165,149.365
C08455=1137.593,-48.787,-46.856,179.140,6.165,149.366
C08456=1137.598,-49.038,-46.846,179.137,6.164,149.366
C08457=1137.604,-49.287,-46.834,179.135,6.163,149.367
C08458=1137.609,-49.537,-46.823,179.133,6.163,149.368
C08459=1137.614,-49.787,-46.812,179.130,6.162,149.368
C08460=1137.620,-50.036,-46.801,179.128,6.161,149.369
C08461=1137.625,-50.286,-46.790,179.125,6.161,149.369
C08462=1137.631,-50.557,-46.779,179.123,6.160,149.370
C08463=1137.636,-50.827,-46.767,179.121,6.160,149.370
C08464=1137.641,-51.098,-46.755,179.118,6.159,149.371
C08465=1137.648,-51.368,-46.743,179.116,6.158,149.372
C08466=1137.653,-51.619,-46.732,179.114,6.158,149.372
C08467=1137.658,-51.868,-46.721,179.111,6.157,149.373
C08468=1137.664,-52.118,-46.710,179.109,6.157,149.373
C08469=1137.668,-52.368,-46.699,179.107,6.156,149.374
C08470=1137.674,-52.617,-46.689,179.105,6.156,149.374
C08471=1137.679,-52.867,-46.677,179.102,6.155,149.375
C08472=1137.684,-53.117,-46.667,179.100,6.155,149.375
C08473=1137.690,-53.366,-46.655,179.098,6.154,149.376
C08474=1137.695,-53.616,-46.645,179.095,6.153,149.377
C08475=1137.700,-53.866,-46.634,179.093,6.153,149.377
C08476=1137.706,-54.115,-46.623,179.091,6.152,149.378
C08477=1137.711,-54.365,-46.613,179.089,6.152,149.378
C08478=1137.715,-54.615,-46.602,179.087,6.151,149.379
C08479=1137.722,-54.865,-46.591,179.084,6.151,149.379
C08480=1137.727,-55.115,-46.580,179.082,6.150,149.380
C08481=1137.732,-55.364,-46.569,179.080,6.150,149.380
C08482=1137.737,-55.614,-46.559,179.077,6.149,149.381
C08483=1137.742,-55.863,-46.548,179.075,6.148,149.381
C08484=1137.747,-56.113,-46.537,179.073,6.147,149.382
C08485=1137.753,-56.363,-46.527,179.071,6.148,149.383
C08486=1137.757,-56.613,-46.516,179.069,6.147,149.383
C08487=1137.763,-56.862,-46.506,179.067,6.146,149.384
C08488=1137.769,-57.113,-46.494,179.064,6.145,149.384
C08489=1137.774,-57.362,-46.483,179.062,6.145,149.385
C08490=1137.779,-57.612,-46.473,179.059,6.144,149.385
C08491=1137.785,-57.861,-46.463,179.057,6.143,149.386
C08492=1137.789,-58.111,-46.451,179.055,6.143,149.386
C08493=1137.795,-58.361,-46.441,179.053,6.143,149.387
C08494=1137.800,-58.611,-46.431,179.051,6.142,149.387
C08495=1137.805,-58.860,-46.420,179.049,6.142,149.388
C08496=1137.810,-59.110,-46.409,179.046,6.141,149.389
C08497=1137.816,-59.360,-46.399,179.044,6.140,149.389
C08498=1137.821,-59.610,-46.388,179.042,6.140,149.389
C08499=1137.826,-59.859,-46.377,179.039,6.139,149.390
C08500=1137.831,-60.109,-46.367,179.037,6.139,149.391
C08501=1137.837,-60.359,-46.357,179.035,6.138,149.391
C08502=1137.842,-60.608,-46.346,179.033,6.138,149.392
C08503=1137.847,-60.858,-46.335,179.030,6.137,149.392
C08504=1137.853,-61.107,-46.325,179.028,6.137,149.393
C08505=1137.858,-61.357,-46.314,179.026,6.136,149.393
C08506=1137.863,-61.607,-46.304,179.024,6.136,149.394
C08507=1137.868,-61.857,-46.293,179.022,6.135,149.394
C08508=1137.874,-62.106,-46.283,179.019,6.135,149.395
C08509=1137.879,-62.356,-46.272,179.017,6.134,149.395
C08510=1137.884,-62.606,-46.262,179.015,6.133,149.396
C08511=1137.890,-62.856,-46.252,179.012,6.133,149.397
C08512=1137.895,-63.106,-46.241,179.011,6.133,149.397
C08513=1137.900,-63.355,-46.230,179.009,6.132,149.398
C08514=1137.905,-63.605,-46.220,179.006,6.131,149.398
C08515=1137.911,-63.854,-46.209,179.004,6.131,149.399
C08516=1137.916,-64.104,-46.199,179.002,6.130,149.399
C08517=1137.921,-64.354,-46.189,178.999,6.129,149.400
C08518=1137.927,-64.604,-46.178,178.998,6.129,149.400
C08519=1137.932,-64.854,-46.168,178.995,6.129,149.401
C08520=1137.937,-65.103,-46.157,178.993,6.128,149.401
C08521=1137.943,-65.353,-46.147,178.991,6.127,149.402
C08522=1137.948,-65.603,-46.136,178.989,6.127,149.402
C08523=1137.953,-65.852,-46.126,178.986,6.126,149.403
C08524=1137.959,-66.102,-46.116,178.984,6.126,149.404
C08525=1137.964,-66.352,-46.105,178.982,6.126,149.404
C08526=1137.969,-66.602,-46.095,178.980,6.125,149.405
C08527=1137.974,-66.852,-46.084,178.977,6.124,149.405
C08528=1137.979,-67.101,-46.075,178.975,6.124,149.406
C08529=1137.985,-67.351,-46.064,178.973,6.124,149.406
C08530=1137.990,-67.601,-46.054,178.971,6.123,149.407
C08531=1137.996,-67.850,-46.044,178.969,6.123,149.407
C08532=1138.001,-68.100,-46.033,178.966,6.122,149.408
C08533=1138.006,-68.350,-46.023,178.964,6.121,149.408
C08534=1138.012,-68.600,-46.013,178.963,6.121,149.409
C08535=1138.017,-68.849,-46.002,178.960,6.121,149.410
C08536=1138.022,-69.099,-45.992,178.958,6.120,149.410
C08537=1138.027,-69.349,-45.982,178.956,6.119,149.411
C08538=1138.033,-69.598,-45.972,178.953,6.118,149.411
C08539=1138.038,-69.849,-45.961,178.951,6.119,149.412
C08540=1138.043,-70.098,-45.951,178.949,6.118,149.412
C08541=1138.049,-70.348,-45.941,178.947,6.117,149.413
C08542=1138.054,-70.597,-45.931,178.945,6.116,149.413
C08543=1138.059,-70.847,-45.921,178.942,6.116,149.414
C08544=1138.064,-71.097,-45.911,178.940,6.116,149.414
C08545=1138.070,-71.346,-45.900,178.938,6.115,149.415
C08546=1138.075,-71.596,-45.890,178.936,6.115,149.415
C08547=1138.081,-71.846,-45.880,178.934,6.114,149.416
C08548=1138.085,-72.095,-45.870,178.931,6.113,149.416
C08549=1138.091,-72.345,-45.861,178.930,6.113,149.417
C08550=1138.096,-72.596,-45.850,178.927,6.113,149.417
C08551=1138.102,-72.845,-45.840,178.925,6.112,149.418
C08552=1138.108,-73.095,-45.830,178.923,6.112,149.419
C08553=1138.112,-73.344,-45.820,178.921,6.112,149.419
C08554=1138.117,-73.594,-45.809,178.919,6.111,149.420
C08555=1138.123,-73.844,-45.799,178.917,6.110,149.420
C08556=1138.129,-74.093,-45.789,178.914,6.110,149.421
C08557=1138.134,-74.343,-45.780,178.912,6.109,149.421
C08558=1138.139,-74.593,-45.770,178.910,6.109,149.422
C08559=1138.144,-74.843,-45.759,178.908,6.108,149.422
C08560=1138.150,-75.093,-45.749,178.906,6.107,149.423
C08561=1138.155,-75.342,-45.739,178.903,6.107,149.423
C08562=1138.160,-75.593,-45.730,178.901,6.107,149.424
C08563=1138.166,-75.842,-45.719,178.899,6.106,149.424
C08564=1138.171,-76.092,-45.709,178.897,6.106,149.425
C08565=1138.176,-76.341,-45.700,178.895,6.105,149.425
C08566=1138.182,-76.613,-45.689,178.892,6.104,149.426
C08567=1138.188,-76.884,-45.678,178.891,6.104,149.427
C08568=1138.194,-77.155,-45.667,178.888,6.104,149.427
C08569=1138.200,-77.427,-45.656,178.886,6.103,149.428
C08570=1138.205,-77.677,-45.646,178.884,6.103,149.428
C08571=1138.210,-77.927,-45.636,178.881,6.102,149.429
C08572=1138.215,-78.177,-45.627,178.879,6.101,149.429
C08573=1138.221,-78.426,-45.617,178.877,6.101,149.430
C08574=1138.226,-78.676,-45.607,178.875,6.101,149.430
C08575=1138.231,-78.925,-45.597,178.873,6.100,149.431
C08576=1138.237,-79.175,-45.587,178.870,6.100,149.432
C08577=1138.242,-79.425,-45.577,178.868,6.100,149.432
C08578=1138.247,-79.675,-45.567,178.866,6.099,149.433
C08579=1138.253,-79.925,-45.558,178.864,6.098,149.433
C08580=1138.258,-80.174,-45.548,178.862,6.097,149.434
C08581=1138.264,-80.424,-45.538,178.860,6.098,149.434
C08582=1138.270,-80.674,-45.528,178.858,6.097,149.435
C08583=1138.274,-80.924,-45.518,178.855,6.096,149.435
C08584=1138.279,-81.173,-45.508,178.854,6.096,149.436
C08585=1138.285,-81.423,-45.499,178.852,6.095,149.436
C08586=1138.290,-81.673,-45.489,178.849,6.095,149.437
C08587=1138.296,-81.922,-45.479,178.847,6.094,149.437
C08588=1138.301,-82.172,-45.470,178.845,6.094,149.438
C08589=1138.306,-82.422,-45.459,178.843,6.094,149.438
C08590=1138.311,-82.672,-45.450,178.841,6.093,149.439
C08591=1138.317,-82.922,-45.440,178.838,6.093,149.440
C08592=1138.322,-83.171,-45.431,178.836,6.093,149.440
C08593=1138.327,-83.421,-45.421,178.834,6.092,149.440
C08594=1138.333,-83.671,-45.411,178.832,6.091,149.441
C08595=1138.338,-83.921,-45.402,178.830,6.091,149.441
C08596=1138.344,-84.170,-45.392,178.828,6.090,149.442
C08597=1138.348,-84.421,-45.382,178.826,6.090,149.443
C08598=1138.354,-84.670,-45.372,178.823,6.089,149.443
C08599=1138.359,-84.920,-45.363,178.822,6.089,149.444
C08600=1138.365,-85.170,-45.353,178.820,6.088,149.444
C08601=1138.370,-85.419,-45.344,178.817,6.088,149.445
C08602=1138.375,-85.669,-45.334,178.815,6.088,149.445
C08603=1138.380,-85.918,-45.324,178.813,6.087,149.446
C08604=1138.386,-86.168,-45.315,178.811,6.087,149.446
C08605=1138.391,-86.418,-45.305,178.809,6.086,149.447
C08606=1138.396,-86.669,-45.295,178.807,6.086,149.447
C08607=1138.401,-86.918,-45.286,178.805,6.085,149.448
C08608=1138.407,-87.168,-45.276,178.802,6.085,149.448
C08609=1138.412,-87.417,-45.267,178.801,6.085,149.449
C08610=1138.418,-87.667,-45.257,178.799,6.084,149.449
C08611=1138.423,-87.917,-45.248,178.796,6.083,149.450
C08612=1138.429,-88.167,-45.238,178.795,6.083,149.450
C08613=1138.434,-88.417,-45.229,178.793,6.083,149.451
C08614=1138.439,-88.666,-45.219,178.790,6.082,149.452
C08615=1138.445,-88.916,-45.210,178.788,6.081,149.452
C08616=1138.450,-89.166,-45.200,178.786,6.081,149.453
C08617=1138.455,-89.415,-45.191,178.784,6.081,149.453
C08618=1138.460,-89.665,-45.181,178.782,6.080,149.453
C08619=1138.466,-89.915,-45.172,178.780,6.080,149.454
C08620=1138.471,-90.165,-45.163,178.777,6.080,149.455
C08621=1138.477,-90.414,-45.153,178.775,6.079,149.455
C08622=1138.482,-90.664,-45.144,178.774,6.079,149.456
C08623=1138.488,-90.914,-45.134,178.771,6.078,149.456
C08624=1138.492,-91.164,-45.124,178.769,6.077,149.457
C08625=1138.497,-91.414,-45.116,178.768,6.077,149.457
C08626=1138.503,-91.664,-45.105,178.765,6.077,149.458
C08627=1138.508,-91.913,-45.096,178.763,6.076,149.458
C08628=1138.514,-92.164,-45.087,178.761,6.076,149.459
C08629=1138.519,-92.413,-45.077,178.759,6.076,149.459
C08630=1138.524,-92.663,-45.068,178.757,6.075,149.460
C08631=1138.530,-92.913,-45.059,178.755,6.075,149.460
C08632=1138.535,-93.162,-45.049,178.753,6.074,149.461
C08633=1138.540,-93.412,-45.040,178.750,6.074,149.461
C08634=1138.546,-93.662,-45.031,178.749,6.074,149.462
C08635=1138.551,-93.911,-45.021,178.747,6.073,149.462
C08636=1138.557,-94.161,-45.012,178.744,6.072,149.463
C08637=1138.562,-94.411,-45.003,178.743,6.072,149.463
C08638=1138.567,-94.661,-44.993,178.741,6.072,149.464
C08639=1138.573,-94.910,-44.984,178.738,6.071,149.464
C08640=1138.578,-95.160,-44.975,178.736,6.071,149.465
C08641=1138.584,-95.410,-44.966,178.734,6.070,149.466
C08642=1138.589,-95.659,-44.956,178.732,6.070,149.466
C08643=1138.594,-95.909,-44.947,178.730,6.070,149.467
C08644=1138.600,-96.159,-44.938,178.728,6.069,149.467
C08645=1138.605,-96.409,-44.929,178.726,6.068,149.467
C08646=1138.611,-96.659,-44.920,178.724,6.068,149.468
C08647=1138.615,-96.908,-44.910,178.722,6.068,149.468
C08648=1138.621,-97.158,-44.901,178.719,6.067,149.469
C08649=1138.627,-97.408,-44.892,178.718,6.067,149.470
C08650=1138.632,-97.658,-44.883,178.716,6.066,149.470
C08651=1138.637,-97.907,-44.873,178.713,6.066,149.471
C08652=1138.642,-98.157,-44.864,178.712,6.066,149.471
C08653=1138.648,-98.407,-44.855,178.710,6.065,149.472
C08654=1138.653,-98.657,-44.846,178.707,6.064,149.472
C08655=1138.658,-98.907,-44.837,178.706,6.064,149.473
C08656=1138.664,-99.156,-44.828,178.703,6.064,149.473
C08657=1138.669,-99.406,-44.819,178.701,6.063,149.474
C08658=1138.674,-99.656,-44.810,178.699,6.063,149.474
C08659=1138.680,-99.905,-44.801,178.697,6.062,149.475
C08660=1138.686,-100.156,-44.791,178.696,6.062,149.475
C08661=1138.691,-100.405,-44.782,178.693,6.062,149.476
C08662=1138.696,-100.655,-44.773,178.691,6.061,149.476
C08663=1138.701,-100.905,-44.765,178.690,6.061,149.477
C08664=1138.707,-101.155,-44.755,178.687,6.060,149.477
C08665=1138.712,-101.404,-44.745,178.685,6.060,149.478
C08666=1138.718,-101.654,-44.737,178.683,6.060,149.478
C08667=1138.723,-101.903,-44.728,178.681,6.059,149.479
C08668=1138.728,-102.153,-44.719,178.679,6.058,149.479
C08669=1138.734,-102.404,-44.710,178.677,6.058,149.480
C08670=1138.740,-102.676,-44.700,178.675,6.058,149.480
C08671=1138.745,-102.948,-44.690,178.672,6.057,149.481
C08672=1138.751,-103.221,-44.680,178.671,6.057,149.482
C08673=1138.756,-103.492,-44.670,178.668,6.057,149.482
C08674=1138.762,-103.742,-44.662,178.666,6.056,149.482
C08675=1138.767,-103.991,-44.653,178.665,6.056,149.483
C08676=1138.773,-104.241,-44.644,178.663,6.055,149.483
C08677=1138.778,-104.491,-44.634,178.660,6.055,149.484
C08678=1138.784,-104.741,-44.625,178.658,6.055,149.485
C08679=1138.789,-104.991,-44.617,178.656,6.054,149.485
C08680=1138.794,-105.241,-44.608,178.654,6.053,149.486
C08681=1138.800,-105.490,-44.599,178.652,6.053,149.486
C08682=1138.805,-105.740,-44.590,178.650,6.053,149.487
C08683=1138.810,-105.990,-44.581,178.648,6.053,149.487
C08684=1138.816,-106.240,-44.572,178.646,6.052,149.488
C08685=1138.821,-106.490,-44.563,178.644,6.051,149.488
C08686=1138.826,-106.740,-44.554,178.642,6.051,149.489
C08687=1138.832,-106.989,-44.546,178.640,6.051,149.489
C08688=1138.837,-107.239,-44.537,178.638,6.051,149.490
C08689=1138.843,-107.489,-44.528,178.636,6.050,149.490
C08690=1138.848,-107.739,-44.520,178.634,6.049,149.491
C08691=1138.853,-107.989,-44.511,178.632,6.050,149.491
C08692=1138.859,-108.238,-44.502,178.630,6.049,149.492
C08693=1138.864,-108.488,-44.493,178.628,6.049,149.492
C08694=1138.869,-108.738,-44.484,178.626,6.048,149.493
C08695=1138.875,-108.988,-44.475,178.624,6.047,149.493
C08696=1138.880,-109.238,-44.466,178.622,6.047,149.494
C08697=1138.886,-109.487,-44.457,178.620,6.047,149.494
C08698=1138.891,-109.737,-44.448,178.619,6.047,149.495
C08699=1138.896,-109.987,-44.440,178.616,6.046,149.495
C08700=1138.902,-110.237,-44.431,178.615,6.046,149.496
C08701=1138.907,-110.486,-44.423,178.613,6.045,149.496
C08702=1138.913,-110.736,-44.414,178.610,6.044,149.497
C08703=1138.918,-110.986,-44.405,178.608,6.045,149.497
C08704=1138.923,-111.236,-44.396,178.606,6.044,149.498
C08705=1138.928,-111.486,-44.387,178.605,6.044,149.498
C08706=1138.934,-111.735,-44.379,178.602,6.043,149.499
C08707=1138.939,-111.985,-44.371,178.600,6.043,149.499
C08708=1138.945,-112.235,-44.362,178.599,6.043,149.500
C08709=1138.950,-112.485,-44.353,178.596,6.042,149.500
C08710=1138.955,-112.734,-44.344,178.595,6.042,149.501
C08711=1138.961,-112.984,-44.335,178.593,6.041,149.501
C08712=1138.966,-113.234,-44.327,178.591,6.041,149.502
C08713=1138.972,-113.484,-44.319,178.589,6.041,149.502
C08714=1138.977,-113.733,-44.310,178.587,6.040,149.503
C08715=1138.982,-113.983,-44.301,178.585,6.040,149.503
C08716=1138.987,-114.233,-44.292,178.583,6.039,149.504
C08717=1138.993,-114.483,-44.284,178.581,6.039,149.504
C08718=1138.999,-114.733,-44.275,178.579,6.038,149.505
C08719=1139.004,-114.983,-44.266,178.577,6.038,149.505
C08720=1139.009,-115.232,-44.257,178.575,6.038,149.506
C08721=1139.015,-115.482,-44.250,178.573,6.037,149.506
C08722=1139.020,-115.732,-44.241,178.571,6.037,149.507
C08723=1139.025,-115.982,-44.232,178.569,6.036,149.507
C08724=1139.031,-116.232,-44.224,178.568,6.036,149.507
C08725=1139.037,-116.482,-44.215,178.565,6.036,149.508
C08726=1139.042,-116.731,-44.206,178.563,6.036,149.509
C08727=1139.048,-116.981,-44.198,178.561,6.035,149.509
C08728=1139.052,-117.231,-44.190,178.560,6.035,149.510
C08729=1139.057,-117.481,-44.181,178.557,6.035,149.510
C08730=1139.063,-117.730,-44.173,178.555,6.034,149.511
C08731=1139.069,-117.980,-44.164,178.554,6.034,149.511
C08732=1139.074,-118.230,-44.156,178.551,6.033,149.512
C08733=1139.080,-118.479,-44.147,178.550,6.033,149.512
C08734=1139.085,-118.730,-44.139,178.548,6.032,149.513
C08735=1139.090,-118.980,-44.130,178.546,6.032,149.513
C08736=1139.096,-119.229,-44.121,178.544,6.032,149.514
C08737=1139.102,-119.479,-44.113,178.542,6.032,149.514
C08738=1139.106,-119.729,-44.105,178.540,6.031,149.515
C08739=1139.112,-119.978,-44.096,178.538,6.030,149.515
C08740=1139.117,-120.228,-44.088,178.536,6.030,149.516
C08741=1139.122,-120.478,-44.079,178.534,6.030,149.516
C08742=1139.128,-120.728,-44.072,178.532,6.030,149.516
C08743=1139.134,-120.978,-44.063,178.530,6.029,149.517
C08744=1139.139,-121.228,-44.054,178.529,6.029,149.517
C08745=1139.144,-121.477,-44.046,178.526,6.028,149.518
C08746=1139.149,-121.727,-44.038,178.525,6.028,149.518
C08747=1139.155,-121.977,-44.029,178.523,6.027,149.519
C08748=1139.160,-122.227,-44.021,178.521,6.028,149.519
C08749=1139.166,-122.477,-44.013,178.519,6.027,149.520
C08750=1139.172,-122.726,-44.004,178.517,6.027,149.520
C08751=1139.176,-122.976,-43.996,178.515,6.026,149.521
C08752=1139.182,-123.226,-43.988,178.513,6.026,149.521
C08753=1139.187,-123.475,-43.979,178.511,6.025,149.522
C08754=1139.193,-123.726,-43.971,178.509,6.025,149.522
C08755=1139.198,-123.976,-43.962,178.507,6.025,149.523
C08756=1139.203,-124.225,-43.955,178.505,6.024,149.523
C08757=1139.209,-124.475,-43.946,178.504,6.024,149.524
C08758=1139.215,-124.725,-43.938,178.501,6.023,149.524
C08759=1139.220,-124.975,-43.929,178.500,6.023,149.525
C08760=1139.225,-125.225,-43.921,178.498,6.023,149.525
C08761=1139.230,-125.474,-43.913,178.496,6.023,149.526
C08762=1139.236,-125.724,-43.905,178.494,6.022,149.526
C08763=1139.242,-125.974,-43.896,178.492,6.022,149.527
C08764=1139.247,-126.224,-43.888,178.490,6.021,149.527
C08765=1139.252,-126.473,-43.880,178.488,6.021,149.528
C08766=1139.257,-126.723,-43.872,178.486,6.020,149.528
C08767=1139.263,-126.973,-43.863,178.485,6.021,149.529
C08768=1139.269,-127.223,-43.855,178.483,6.019,149.529
C08769=1139.273,-127.472,-43.847,178.481,6.019,149.529
C08770=1139.279,-127.722,-43.839,178.479,6.019,149.530
C08771=1139.285,-127.973,-43.831,178.478,6.019,149.530
C08772=1139.290,-128.222,-43.823,178.475,6.018,149.531
C08773=1139.295,-128.472,-43.815,178.474,6.018,149.531
C08774=1138.875,-128.483,-43.858,178.470,6.021,149.533
C08775=1138.869,-128.234,-43.866,178.472,6.022,149.533
C08776=1138.863,-127.983,-43.874,178.474,6.022,149.532
C08777=1138.858,-127.733,-43.883,178.476,6.023,149.532
C08778=1138.853,-127.484,-43.891,178.478,6.023,149.531
C08779=1138.848,-127.234,-43.900,178.480,6.023,149.531
C08780=1138.842,-126.984,-43.907,178.481,6.023,149.530
C08781=1138.837,-126.735,-43.916,178.484,6.024,149.530
C08782=1138.831,-126.485,-43.923,178.485,6.024,149.529
C08783=1138.826,-126.234,-43.932,178.487,6.025,149.529
C08784=1138.820,-125.985,-43.941,178.489,6.025,149.528
C08785=1138.815,-125.735,-43.948,178.491,6.026,149.528
C08786=1138.810,-125.485,-43.957,178.493,6.025,149.527
C08787=1138.804,-125.236,-43.964,178.495,6.026,149.527
C08788=1138.799,-124.986,-43.973,178.496,6.026,149.526
C08789=1138.793,-124.736,-43.981,178.499,6.027,149.526
C08790=1138.788,-124.486,-43.989,178.500,6.027,149.525
C08791=1138.783,-124.236,-43.998,178.502,6.028,149.525
C08792=1138.777,-123.987,-44.006,178.504,6.028,149.525
C08793=1138.771,-123.736,-44.014,178.506,6.029,149.524
C08794=1138.766,-123.487,-44.023,178.508,6.029,149.524
C08795=1138.761,-123.238,-44.031,178.510,6.029,149.523
C08796=1138.756,-122.987,-44.039,178.512,6.030,149.523
C08797=1138.750,-122.738,-44.048,178.513,6.030,149.522
C08798=1138.745,-122.488,-44.056,178.516,6.031,149.522
C08799=1138.739,-122.238,-44.065,178.517,6.031,149.521
C08800=1138.734,-121.988,-44.072,178.519,6.032,149.521
C08801=1138.729,-121.738,-44.081,178.521,6.031,149.520
C08802=1138.723,-121.489,-44.089,178.523,6.032,149.520
C08803=1138.718,-121.239,-44.098,178.525,6.032,149.519
C08804=1138.713,-120.989,-44.107,178.527,6.033,149.519
C08805=1138.706,-120.739,-44.115,178.529,6.033,149.518
C08806=1138.702,-120.490,-44.123,178.531,6.034,149.518
C08807=1138.697,-120.239,-44.131,178.532,6.034,149.517
C08808=1138.691,-119.990,-44.140,178.535,6.034,149.517
C08809=1138.686,-119.740,-44.148,178.537,6.035,149.516
C08810=1138.680,-119.490,-44.157,178.538,6.035,149.516
C08811=1138.674,-119.240,-44.165,178.541,6.036,149.515
C08812=1138.669,-118.991,-44.174,178.542,6.036,149.515
C08813=1138.664,-118.740,-44.182,178.544,6.036,149.514
C08814=1138.659,-118.491,-44.190,178.546,6.036,149.514
C08815=1138.654,-118.241,-44.199,178.548,6.037,149.513
C08816=1138.648,-117.991,-44.207,178.550,6.037,149.513
C08817=1138.642,-117.742,-44.216,178.552,6.038,149.512
C08818=1138.637,-117.492,-44.225,178.554,6.037,149.512
C08819=1138.632,-117.242,-44.233,178.556,6.038,149.511
C08820=1138.626,-116.992,-44.241,178.558,6.039,149.511
C08821=1138.621,-116.743,-44.250,178.560,6.039,149.510
C08822=1138.615,-116.492,-44.259,178.562,6.040,149.510
C08823=1138.609,-116.243,-44.267,178.564,6.040,149.509
C08824=1138.604,-115.993,-44.276,178.566,6.040,149.509
C08825=1138.599,-115.743,-44.285,178.568,6.040,149.508
C08826=1138.593,-115.493,-44.293,178.570,6.041,149.508
C08827=1138.589,-115.244,-44.301,178.572,6.042,149.507
C08828=1138.583,-114.994,-44.310,178.574,6.042,149.507
C08829=1138.578,-114.744,-44.319,178.576,6.042,149.506
C08830=1138.572,-114.494,-44.327,178.577,6.042,149.506
C08831=1138.567,-114.245,-44.335,178.580,6.043,149.505
C08832=1138.562,-113.995,-44.344,178.581,6.043,149.505
C08833=1138.556,-113.746,-44.353,178.583,6.044,149.504
C08834=1138.551,-113.495,-44.361,178.586,6.045,149.504
C08835=1138.545,-113.245,-44.370,178.587,6.045,149.503
C08836=1138.540,-112.995,-44.379,178.589,6.045,149.503
C08837=1138.535,-112.746,-44.387,178.591,6.045,149.503
C08838=1138.529,-112.496,-44.396,178.593,6.046,149.502
C08839=1138.524,-112.246,-44.404,178.595,6.046,149.502
C08840=1138.519,-111.996,-44.413,178.597,6.047,149.501
C08841=1138.513,-111.747,-44.422,178.599,6.047,149.501
C08842=1138.508,-111.497,-44.431,178.601,6.047,149.500
C08843=1138.503,-111.247,-44.440,178.603,6.048,149.500
C08844=1138.497,-110.997,-44.448,178.605,6.048,149.499
C08845=1138.491,-110.748,-44.456,178.607,6.048,149.498
C08846=1138.486,-110.498,-44.465,178.609,6.048,149.498
C08847=1138.480,-110.248,-44.475,178.611,6.049,149.497
C08848=1138.475,-109.998,-44.484,178.613,6.050,149.497
C08849=1138.470,-109.748,-44.493,178.615,6.050,149.496
C08850=1138.464,-109.499,-44.501,178.617,6.051,149.496
C08851=1138.459,-109.249,-44.510,178.619,6.051,149.495
C08852=1138.454,-108.998,-44.518,178.621,6.051,149.495
C08853=1138.448,-108.749,-44.527,178.623,6.052,149.494
C08854=1138.443,-108.499,-44.536,178.625,6.052,149.494
C08855=1138.438,-108.250,-44.545,178.627,6.053,149.494
C08856=1138.432,-108.000,-44.553,178.628,6.053,149.493
C08857=1138.427,-107.750,-44.562,178.631,6.054,149.493
C08858=1138.422,-107.500,-44.571,178.633,6.054,149.492
C08859=1138.417,-107.250,-44.580,178.634,6.054,149.492
C08860=1138.411,-107.001,-44.589,178.637,6.055,149.491
C08861=1138.405,-106.751,-44.598,178.639,6.055,149.490
C08862=1138.400,-106.501,-44.607,178.641,6.055,149.490
C08863=1138.395,-106.251,-44.616,178.643,6.056,149.489
C08864=1138.390,-106.001,-44.625,178.645,6.056,149.489
C08865=1138.384,-105.752,-44.633,178.647,6.057,149.488
C08866=1138.379,-105.502,-44.642,178.648,6.057,149.488
C08867=1138.374,-105.252,-44.651,178.651,6.057,149.487
C08868=1138.368,-105.003,-44.660,178.653,6.058,149.487
C08869=1138.363,-104.752,-44.670,178.654,6.058,149.486
C08870=1138.357,-104.503,-44.678,178.657,6.059,149.486
C08871=1138.352,-104.253,-44.687,178.659,6.060,149.485
C08872=1138.346,-104.004,-44.696,178.661,6.059,149.485
C08873=1138.341,-103.754,-44.705,178.663,6.060,149.484
C08874=1138.336,-103.504,-44.714,178.665,6.060,149.484
C08875=1138.330,-103.231,-44.723,178.667,6.061,149.483
C08876=1138.325,-102.959,-44.733,178.669,6.061,149.483
C08877=1138.318,-102.687,-44.744,178.672,6.062,149.482
C08878=1138.312,-102.414,-44.753,178.673,6.062,149.482
C08879=1138.307,-102.165,-44.762,178.676,6.063,149.481
C08880=1138.302,-101.916,-44.771,178.678,6.063,149.481
C08881=1138.297,-101.666,-44.780,178.679,6.063,149.480
C08882=1138.291,-101.416,-44.789,178.682,6.064,149.480
C08883=1138.286,-101.166,-44.798,178.684,6.065,149.479
C08884=1138.280,-100.916,-44.807,178.685,6.065,149.479
C08885=1138.275,-100.666,-44.816,178.688,6.065,149.478
C08886=1138.270,-100.416,-44.825,178.690,6.065,149.478
C08887=1138.264,-100.166,-44.835,178.692,6.066,149.477
C08888=1138.258,-99.917,-44.843,178.694,6.067,149.477
C08889=1138.254,-99.668,-44.853,178.696,6.066,149.476
C08890=1138.248,-99.418,-44.862,178.698,6.067,149.476
C08891=1138.242,-99.168,-44.871,178.700,6.068,149.475
C08892=1138.237,-98.918,-44.880,178.702,6.068,149.475
C08893=1138.232,-98.668,-44.889,178.704,6.069,149.474
C08894=1138.227,-98.418,-44.898,178.706,6.069,149.473
C08895=1138.221,-98.169,-44.908,178.708,6.069,149.473
C08896=1138.216,-97.919,-44.917,178.710,6.070,149.472
C08897=1138.211,-97.669,-44.926,178.712,6.071,149.472
C08898=1138.205,-97.419,-44.935,178.714,6.070,149.471
C08899=1138.200,-97.169,-44.944,178.716,6.071,149.471
C08900=1138.195,-96.920,-44.954,178.718,6.071,149.471
C08901=1138.189,-96.670,-44.962,178.720,6.072,149.470
C08902=1138.183,-96.420,-44.972,178.723,6.072,149.469
C08903=1138.178,-96.170,-44.981,178.724,6.072,149.469
C08904=1138.173,-95.921,-44.990,178.726,6.073,149.468
C08905=1138.168,-95.671,-45.000,178.729,6.074,149.468
C08906=1138.162,-95.421,-45.009,178.730,6.074,149.467
C08907=1138.157,-95.171,-45.018,178.732,6.074,149.467
C08908=1138.151,-94.921,-45.027,178.735,6.075,149.466
C08909=1138.146,-94.672,-45.037,178.736,6.075,149.466
C08910=1138.141,-94.422,-45.046,178.739,6.076,149.465
C08911=1138.135,-94.172,-45.055,178.741,6.076,149.465
C08912=1138.130,-93.923,-45.065,178.743,6.076,149.464
C08913=1138.125,-93.673,-45.074,178.745,6.077,149.464
C08914=1138.119,-93.423,-45.083,178.747,6.078,149.463
C08915=1138.114,-93.173,-45.092,178.749,6.078,149.463
C08916=1138.109,-92.924,-45.102,178.751,6.079,149.462
C08917=1138.103,-92.673,-45.111,178.754,6.079,149.462
C08918=1138.098,-92.424,-45.120,178.755,6.079,149.461
C08919=1138.093,-92.174,-45.130,178.757,6.080,149.461
C08920=1138.088,-91.924,-45.139,178.760,6.080,149.460
C08921=1138.082,-91.674,-45.148,178.761,6.080,149.460
C08922=1138.077,-91.425,-45.158,178.763,6.081,149.459
C08923=1138.072,-91.175,-45.167,178.766,6.082,149.459
C08924=1138.066,-90.925,-45.177,178.768,6.082,149.458
C08925=1138.061,-90.676,-45.186,178.770,6.082,149.457
C08926=1138.056,-90.426,-45.195,178.772,6.083,149.457
C08927=1138.050,-90.176,-45.205,178.774,6.084,149.456
C08928=1138.045,-89.926,-45.214,178.776,6.084,149.456
C08929=1138.039,-89.676,-45.224,178.778,6.084,149.456
C08930=1138.034,-89.427,-45.233,178.781,6.085,149.455
C08931=1138.028,-89.177,-45.243,178.782,6.085,149.454
C08932=1138.023,-88.928,-45.253,178.784,6.085,149.454
C08933=1138.017,-88.677,-45.262,178.787,6.086,149.453
C08934=1138.013,-88.428,-45.272,178.788,6.086,149.453
C08935=1138.008,-88.178,-45.281,178.790,6.087,149.452
C08936=1138.002,-87.928,-45.291,178.793,6.087,149.452
C08937=1137.997,-87.678,-45.300,178.795,6.088,149.451
C08938=1137.991,-87.428,-45.310,178.797,6.088,149.451
C08939=1137.987,-87.179,-45.319,178.799,6.089,149.450
C08940=1137.981,-86.929,-45.329,178.801,6.090,149.450
C08941=1137.976,-86.679,-45.338,178.803,6.090,149.449
C08942=1137.970,-86.429,-45.348,178.806,6.090,149.449
C08943=1137.965,-86.180,-45.357,178.808,6.091,149.448
C08944=1137.959,-85.930,-45.367,178.809,6.091,149.448
C08945=1137.954,-85.681,-45.376,178.812,6.091,149.447
C08946=1137.948,-85.430,-45.386,178.814,6.092,149.447
C08947=1137.944,-85.181,-45.396,178.816,6.093,149.446
C08948=1137.938,-84.931,-45.406,178.818,6.092,149.445
C08949=1137.933,-84.681,-45.415,178.820,6.093,149.445
C08950=1137.928,-84.432,-45.425,178.822,6.094,149.444
C08951=1137.923,-84.182,-45.434,178.824,6.094,149.444
C08952=1137.917,-83.932,-45.444,178.826,6.095,149.443
C08953=1137.912,-83.682,-45.453,178.828,6.095,149.443
C08954=1137.906,-83.433,-45.463,178.831,6.096,149.442
C08955=1137.901,-83.182,-45.473,178.833,6.096,149.442
C08956=1137.896,-82.933,-45.483,178.835,6.097,149.441
C08957=1137.890,-82.683,-45.493,178.837,6.097,149.441
C08958=1137.885,-82.433,-45.502,178.839,6.098,149.440
C08959=1137.880,-82.184,-45.512,178.841,6.098,149.440
C08960=1137.874,-81.934,-45.522,178.843,6.098,149.439
C08961=1137.869,-81.684,-45.531,178.846,6.099,149.439
C08962=1137.863,-81.435,-45.542,178.847,6.099,149.438
C08963=1137.859,-81.184,-45.551,178.849,6.100,149.438
C08964=1137.853,-80.935,-45.561,178.852,6.100,149.437
C08965=1137.848,-80.685,-45.571,178.854,6.101,149.437
C08966=1137.842,-80.435,-45.580,178.856,6.101,149.436
C08967=1137.837,-80.186,-45.590,178.858,6.102,149.436
C08968=1137.832,-79.937,-45.600,178.860,6.103,149.435
C08969=1137.827,-79.686,-45.610,178.863,6.103,149.434
C08970=1137.821,-79.436,-45.620,178.865,6.103,149.434
C08971=1137.816,-79.187,-45.630,178.867,6.104,149.433
C08972=1137.810,-78.937,-45.639,178.869,6.104,149.433
C08973=1137.805,-78.687,-45.649,178.871,6.105,149.432
C08974=1137.800,-78.437,-45.659,178.873,6.105,149.432
C08975=1137.795,-78.188,-45.670,178.875,6.105,149.431
C08976=1137.789,-77.938,-45.679,178.878,6.106,149.431
C08977=1137.784,-77.688,-45.689,178.880,6.107,149.430
C08978=1137.778,-77.439,-45.699,178.881,6.107,149.430
C08979=1137.773,-77.167,-45.709,178.884,6.107,149.429
C08980=1137.767,-76.895,-45.721,178.886,6.108,149.429
C08981=1137.761,-76.624,-45.731,178.889,6.108,149.428
C08982=1137.755,-76.352,-45.742,178.891,6.109,149.427
C08983=1137.750,-76.103,-45.752,178.893,6.110,149.427
C08984=1137.745,-75.853,-45.762,178.896,6.111,149.426
C08985=1137.739,-75.603,-45.772,178.898,6.110,149.426
C08986=1137.734,-75.353,-45.782,178.900,6.111,149.425
C08987=1137.729,-75.104,-45.792,178.902,6.112,149.425
C08988=1137.723,-74.854,-45.802,178.904,6.113,149.424
C08989=1137.718,-74.604,-45.812,178.906,6.113,149.424
C08990=1137.713,-74.355,-45.823,178.908,6.113,149.423
C08991=1137.707,-74.105,-45.831,178.911,6.114,149.423
C08992=1137.702,-73.855,-45.842,178.913,6.114,149.422
C08993=1137.697,-73.605,-45.852,178.914,6.114,149.422
C08994=1137.691,-73.355,-45.862,178.917,6.115,149.421
C08995=1137.686,-73.106,-45.872,178.919,6.116,149.420
C08996=1137.681,-72.857,-45.882,178.921,6.116,149.420
C08997=1137.675,-72.606,-45.892,178.924,6.117,149.419
C08998=1137.670,-72.356,-45.902,178.925,6.117,149.419
C08999=1137.664,-72.107,-45.913,178.928,6.117,149.418
C09000=1137.659,-71.858,-45.922,178.930,6.118,149.418
C09001=1137.654,-71.607,-45.933,178.932,6.119,149.417
C09002=1137.649,-71.358,-45.943,178.934,6.119,149.417
C09003=1137.643,-71.108,-45.953,178.937,6.119,149.416
C09004=1137.638,-70.858,-45.964,178.939,6.120,149.416
C09005=1137.633,-70.609,-45.973,178.941,6.121,149.415
C09006=1137.628,-70.359,-45.984,178.943,6.122,149.415
C09007=1137.623,-70.109,-45.994,178.945,6.122,149.414
C09008=1137.617,-69.859,-46.004,178.947,6.122,149.414
C09009=1137.612,-69.610,-46.015,178.950,6.123,149.413
C09010=1137.606,-69.360,-46.025,178.952,6.123,149.413
C09011=1137.601,-69.110,-46.035,178.954,6.124,149.412
C09012=1137.596,-68.861,-46.045,178.956,6.124,149.411
C09013=1137.590,-68.611,-46.054,178.958,6.125,149.411
C09014=1137.585,-68.360,-46.065,178.960,6.125,149.410
C09015=1137.580,-68.112,-46.076,178.963,6.126,149.410
C09016=1137.574,-67.862,-46.086,178.965,6.126,149.409
C09017=1137.569,-67.612,-46.097,178.967,6.126,149.409
C09018=1137.564,-67.362,-46.107,178.969,6.127,149.408
C09019=1137.558,-67.113,-46.117,178.971,6.128,149.408
C09020=1137.554,-66.863,-46.127,178.974,6.128,149.407
C09021=1137.548,-66.613,-46.137,178.976,6.129,149.407
C09022=1137.543,-66.363,-46.148,178.978,6.130,149.406
C09023=1137.538,-66.113,-46.158,178.980,6.130,149.406
C09024=1137.532,-65.864,-46.168,178.983,6.130,149.405
C09025=1137.527,-65.614,-46.179,178.985,6.131,149.404
C09026=1137.521,-65.364,-46.189,178.987,6.132,149.404
C09027=1137.516,-65.114,-46.199,178.989,6.133,149.403
C09028=1137.511,-64.864,-46.210,178.991,6.132,149.403
C09029=1137.505,-64.615,-46.220,178.993,6.133,149.402
C09030=1137.500,-64.364,-46.231,178.996,6.134,149.402
C09031=1137.495,-64.116,-46.242,178.998,6.134,149.401
C09032=1137.489,-63.866,-46.252,179.001,6.135,149.401
C09033=1137.484,-63.616,-46.262,179.003,6.136,149.400
C09034=1137.480,-63.367,-46.272,179.004,6.136,149.400
C09035=1137.475,-63.116,-46.283,179.006,6.136,149.399
C09036=1137.469,-62.867,-46.293,179.009,6.137,149.398
C09037=1137.464,-62.618,-46.304,179.011,6.137,149.398
C09038=1137.459,-62.368,-46.314,179.014,6.138,149.397
C09039=1137.453,-62.118,-46.324,179.016,6.139,149.397
C09040=1137.448,-61.868,-46.335,179.018,6.139,149.396
C09041=1137.442,-61.618,-46.345,179.020,6.139,149.396
C09042=1137.437,-61.368,-46.356,179.022,6.140,149.395
C09043=1137.432,-61.119,-46.367,179.024,6.141,149.395
C09044=1137.427,-60.870,-46.377,179.027,6.141,149.394
C09045=1137.422,-60.619,-46.388,179.029,6.142,149.394
C09046=1137.416,-60.370,-46.398,179.031,6.142,149.393
C09047=1137.411,-60.120,-46.409,179.033,6.143,149.393
C09048=1137.405,-59.870,-46.420,179.036,6.143,149.392
C09049=1137.400,-59.620,-46.430,179.038,6.144,149.392
C09050=1137.394,-59.370,-46.441,179.040,6.145,149.391
C09051=1137.390,-59.121,-46.452,179.042,6.146,149.391
C09052=1137.384,-58.871,-46.462,179.045,6.146,149.390
C09053=1137.379,-58.621,-46.473,179.047,6.146,149.389
C09054=1137.374,-58.372,-46.484,179.049,6.147,149.389
C09055=1137.369,-58.122,-46.494,179.051,6.147,149.388
C09056=1137.363,-57.872,-46.504,179.054,6.148,149.388
C09057=1137.358,-57.623,-46.515,179.056,6.149,149.387
C09058=1137.353,-57.373,-46.526,179.058,6.149,149.387
C09059=1137.347,-57.124,-46.536,179.061,6.150,149.386
C09060=1137.342,-56.873,-46.547,179.063,6.150,149.386
C09061=1137.337,-56.624,-46.558,179.064,6.150,149.385
C09062=1137.331,-56.374,-46.569,179.067,6.151,149.385
C09063=1137.327,-56.124,-46.580,179.069,6.152,149.384
C09064=1137.321,-55.875,-46.590,179.071,6.152,149.383
C09065=1137.316,-55.624,-46.601,179.074,6.153,149.383
C09066=1137.311,-55.376,-46.612,179.076,6.154,149.382
C09067=1137.306,-55.125,-46.622,179.078,6.154,149.382
C09068=1137.300,-54.876,-46.633,179.081,6.155,149.381
C09069=1137.295,-54.626,-46.644,179.082,6.155,149.381
C09070=1137.289,-54.376,-46.655,179.085,6.155,149.380
C09071=1137.284,-54.127,-46.666,179.087,6.156,149.380
C09072=1137.279,-53.877,-46.676,179.089,6.157,149.379
C09073=1137.274,-53.628,-46.687,179.092,6.157,149.378
C09074=1137.268,-53.378,-46.698,179.094,6.158,149.378
C09075=1137.263,-53.128,-46.708,179.096,6.159,149.377
C09076=1137.257,-52.878,-46.720,179.099,6.160,149.377
C09077=1137.252,-52.628,-46.730,179.101,6.160,149.376
C09078=1137.248,-52.379,-46.742,179.103,6.160,149.376
C09079=1137.242,-52.129,-46.752,179.105,6.161,149.375
C09080=1137.237,-51.879,-46.763,179.108,6.161,149.375
C09081=1137.231,-51.630,-46.774,179.110,6.162,149.374
C09082=1137.226,-51.380,-46.785,179.112,6.163,149.374
C09083=1137.221,-51.109,-46.797,179.115,6.163,149.373
C09084=1137.215,-50.838,-46.808,179.117,6.164,149.373
C09085=1137.209,-50.567,-46.820,179.120,6.164,149.372
C09086=1137.203,-50.297,-46.832,179.122,6.165,149.371
C09087=1137.198,-50.048,-46.843,179.124,6.166,149.371
C09088=1137.193,-49.797,-46.854,179.127,6.166,149.370
C09089=1137.187,-49.548,-46.866,179.129,6.167,149.370
C09090=1137.182,-49.298,-46.876,179.131,6.168,149.369
C09091=1137.177,-49.049,-46.887,179.134,6.168,149.368
C09092=1137.172,-48.799,-46.899,179.136,6.169,149.368
C09093=1137.167,-48.549,-46.909,179.138,6.170,149.368
C09094=1137.161,-48.300,-46.920,179.140,6.171,149.367
C09095=1137.156,-48.050,-46.931,179.142,6.170,149.366
C09096=1137.151,-47.800,-46.943,179.145,6.171,149.366
C09097=1137.146,-47.551,-46.954,179.147,6.172,149.365
C09098=1137.141,-47.300,-46.964,179.149,6.172,149.365
C09099=1137.135,-47.051,-46.976,179.152,6.173,149.364
C09100=1137.130,-46.801,-46.986,179.154,6.174,149.364
C09101=1137.125,-46.551,-46.998,179.156,6.174,149.363
C09102=1137.119,-46.302,-47.009,179.159,6.175,149.363
C09103=1137.114,-46.052,-47.020,179.161,6.176,149.362
C09104=1137.109,-45.802,-47.031,179.163,6.176,149.362
C09105=1137.103,-45.553,-47.043,179.166,6.177,149.361
C09106=1137.098,-45.303,-47.053,179.168,6.177,149.360
C09107=1137.094,-45.053,-47.065,179.170,6.178,149.360
C09108=1137.088,-44.804,-47.076,179.173,6.179,149.359
C09109=1137.083,-44.554,-47.087,179.175,6.179,149.359
C09110=1137.077,-44.304,-47.098,179.176,6.179,149.358
C09111=1137.072,-44.055,-47.109,179.179,6.180,149.358
C09112=1137.067,-43.805,-47.121,179.181,6.181,149.357
